(* IEC 61131-3 sources: NachHouse_CORE/V200/APP (part 3) *)

		r2	: NH_DAT_TIM2  := (txt:=                        	// zadanie datumu/casu
         [ (),(),(),(),(),(),(),(),
				(wh:=0),             										// ziadny text v urovni title
				(wh:=0)                         							// ziadny text pred datumom
			]);

      s  	: ARRAY[0..1] OF NH_SLD_DAT :=
         [  (t:=1,v1:=1, v2:=31, fmt := '%3.0f', txt:= 116, zom:=0,tun:=0),        										// 0 slider k start
				(t := 5,v1:=1,       v2 := 1439.0  , fmt := ''          , txt :=   0, xv := x2-53, tun := 1  )    // slider LUPY bodu, nevypisuje sa ani text, ani hodnota
         ];
   END_STRUCT;
  	NH_FRM_031  {HIDDEN} :    STRUCT     //31 FRM - ROM*set typ miestnosti
      hed : NH_FRM_HED := (Name:='_031',wht:=2,row:=1,sld:=0,desc:='Typ ROM');
      txt   : ARRAY[0..0] OF NH_OBJ_DAT :=
          [(wh:=6 , x:=xc,       y:= y1 + 60,  w:= 400, h:=28, Fgc:=4, fn:=2, nTch:=1, cf:=(n:=435))];           // typ miestosti

      mnu   : NH_OBJ_123 := // 2 riadky
            (wh:=123,cf:=(x:= 100,     y:= y1 + 130, typ:=2, rw2:=7, h:= 50, hTxt:= 28),
                 txt:=[436,437,438,439,440,441,511,512]);                                                    // 1 rolovaci vyber textov
      wrk   : ARRAY[3..10] OF NH_OBJ_DAT :=
          [(wh:= 0,   x:= xc , 		y:= y1 + 690, w:= 450, Fn := 2,  FgC :=5, BgC := 0, h := 24, cf:=(c:=0,n:=563), nTch:=1),	// 3 pouzit snimac osvelenia z
           (wh:=21,  x:= x2- 70 , 	y:= y1 + 550,  w:= 45, Fn :=563, FgC := 4, BgC := 50, h:=26),    	// 4 teplotu zo zony
           (wh:= 0,  x:= x2- 70 , 	y:= y1 + 600,  w:= 45, Fn :=564, FgC := 4, BgC := 50, h:=26),     // 5 osvetlenie z vonkajsej zony
           (wh:= 0,  x:= x2- 70 , 	y:= y1 + 650,  w:= 45, Fn :=565, FgC := 4, BgC := 50, h:=26),     // 6 osvetlenie z nadradenej zony
           (wh:=21,  x:= x2- 70 , 	y:= y1 + 700,  w:= 45, Fn :=566, FgC := 4, BgC := 50, h:=26),      // 7 CO2 zo zony
           (wh:= 0,  x:= x2- 70 , 	y:= y1 + 830,  w:= 45, Fn :=566, FgC := 4, BgC := 50, h:=26),
           (wh:= 0,  x:= x2- 70 , 	y:= y1 + 875,  w:= 45, Fn :=567, FgC := 4, BgC := 50, h:=26)
				// pred 3

			];

   END_STRUCT

//   NH_ZON_SET  {HIDDEN} : STRUCT      // ROM typ miestnosti
  	NH_FRM_032  {HIDDEN} :    STRUCT              //32 FRM - ZON*Set typ zony ....
      hed : NH_FRM_HED := (Name:='_032',wht:=2,row:=1,sld:=0,desc:='Typ ZON');

      txt   : ARRAY[0..0] OF NH_OBJ_DAT :=
          [ (wh:=6 , x:=xc,       y:= y1 + 60,  w:= 400, h:=28, Fgc:=4, fn:=2, nTch:=1, cf:=(n:=442))];           // typ miestosti
      mnu   : NH_OBJ_123 := // 2 riadky
            (wh:=123,cf:=(x:= 100,     y:= y1 + 130, typ:=2, rw2:=5, h:= 50, hTxt:= 28),
                 txt:=[443,444,445,446,447]);                                                    // 1 rolovaci vyber textov
      wrk   : ARRAY[3..10] OF NH_OBJ_DAT :=
          [(wh:= 0,  x:= xc , 		y:= y1 + 690, w:= 450, Fn := 2,  FgC :=5, BgC := 0, h := 24, cf:=(c:=0,n:=563), nTch:=1),	// 3 pouzit snimac osvelenia z
           (wh:= 0,  x:= x2- 70 , 	y:= y1 + 740,  w:= 45, Fn :=564, FgC := 4, BgC := 50, h:=22),                                    // 4
           (wh:= 0,  x:= x2- 70 , 	y:= y1 + 785,  w:= 45, Fn :=565, FgC := 4, BgC := 50, h:=22),
           (wh:= 0,  x:= x2- 70 , 	y:= y1 + 830,  w:= 45, Fn :=566, FgC := 4, BgC := 50, h:=22),
           (wh:= 0,  x:= x2- 70 , 	y:= y1 + 875,  w:= 45, Fn :=567, FgC := 4, BgC := 50, h:=22)
			];
   END_STRUCT

   NH_FRM_033  {HIDDEN} :  STRUCT 	// FRM - predvlby teploty
      hed : NH_FRM_HED := (Name:='_033',wht:=2,row:=1,sld:=5);
		PV_0_2			: ARRAY[0..2] OF NH_OBJ_DAT;
 		TX2				: NH_OBJ_DAT :=
		 		(wh:=6,  x:= x2/2   , 	y:= y1 +250, w:= 400,FgC := 4, BgC := 0, fn := 2, 	h:=33,cf:=(n:=592));   		// predvolby reguluju
		PV_4_10			: ARRAY[4..10] OF NH_OBJ_DAT;

      PV_SLD_XXX  	: ARRAY[0..4] OF NH_SLD_DAT :=  // definica a nazvy sliderov
         [  (t:=0,	xv := x2-53, v1 := 0.0, v2 :=100.0 , fmt := '%5.0f %%'       			   ,txt:= 83 ),     // 0 off       	txt:=cislo textu
            (t:=0,	xv := x2-53, v1 := 0.0, v2 :=100.0 , fmt := '%5.0f %%'      			   ,txt:= 154),     // 1 Minimum
            (t:=0,	xv := x2-53, v1 := 0.0, v2 :=100.0 , fmt := '%5.0f %%'      			   ,txt:= 156),     // 2 Normal
            (t:=0,	xv := x2-53, v1 := 0.0, v2 :=100.0 , fmt := '%5.0f %%'						,txt:= 165),     // 3 Maximum
            (t:=1, 	xv := x2-53, v2 :=255.0, 				 fmt := 's%Tm:ss m'						,txt:= 190) 	  // 4 opozdenie technologie
			];

   END_STRUCT;

	NH_FRM_035  {HIDDEN}  :  STRUCT 	//
      hed : NH_FRM_HED := (Name:='_035',desc:='FRM-TER/TEH/TEK Stp',wht:=2,row:=1,sld:=4);
      r  : ARRAY[1..1] OF NH_ROW_O := [( ob := [
            (wh:=221,x:= 50	,y:= y1 + 100, w:= 25 , 	h := 30,  	FgC :=10, BgC := 5,	Fn :=132,),     			// 0 hodnota zo snimaca
            (wh:=13, x:= 50   ,y:= y1 + 220, w:= x2-110, h := 251,	FgC := 4, BgC := 3, 	fn := 0),            	// 1 Korekcia - Konverzý faktor
            (wh:=221,x:= 50	,y:= y1 + 310, w:= 25 , 	h := 30,  	FgC := 3, BgC := 5, 	fn :=149,),          	// 2 hodnota po korekcii
           	(),
            (),
            (),
            (wh:=13, x:= 50   ,y:= y1 + 500, w:= x2-110 , h := 251,	FgC := 4, BgC := 2, 	fn := 1),              	// 6 povolena zmena
            (wh:=13, x:= 50   ,y:= y1 + 600, w:= x2-110 , h := 251,	FgC := 4, BgC := 2, 	fn := 2),              	// 7 opozdnie zmeny
            (wh:=13, x:= 50   ,y:= y1 + 700, w:= x2-110 , h := 251,	FgC := 4, BgC := 2, 	fn := 3),              	// 8
			   (wh:=20, x:=x2-60 ,y:= y1 + 820, w:= 48     , 				FgC := 0, BgC :=50, 	fn := 241),	  				// 9 neposielat do room
			   (wh:=20, x:=x2-60 ,y:= y1 + 880, w:= 48     , 				FgC := 4, BgC :=50, 	fn := 100)  				//10 zablokovat

       )];
      s  : ARRAY[0..3] OF NH_SLD_DAT := [
            ( t:=0, xv := x2-53, v1:=-20.0, 	v2 := 20.0 ,  fmt := '%+5.1f °C',   txt:= 119, ink:=0.1),      	// 0 Korekcia - Konverzý faktor
            ( t:=0, xv := x2-53, v1:=0.0, 	v2 := 10.0 ,  fmt := '%5.1f', 		txt:= 121, ink:=0.1),			// 1 povolena zmena
            ( t:=1, xv := x2-53, v1:=0.0, 	v2 := 254.0 , fmt := '%5.0f',   		txt:= 122),      					// 2 opozdenie zmeny
            ( t:=3, xv := x2-53, v1:=0.0, 	v2 := 3600.0, fmt := 's%Th:mm:ss h', 	txt:= 609)       					// 3 odoberat vzorky
			];
   END_STRUCT;

   NH_FRM_036 {HIDDEN}  :  STRUCT
      hed      : NH_FRM_HED := (Name:='_036',wht:=3);
      mnu      : NH_MNU := ( n:= 3,        // 7 MNU - TVE/VEN
                        o := [
                              (fn :=  6,wh:=   0,cm := 136),       		// < 1
                              (fn := 183,wh:= 25,cm :=   0),       		// 2
                              (fn := 344,wh:=345,cm := 205, frm:=33),  	// 3-predvolby
                              (fn := 220,wh:=221,cm := 205, frm:=30),   // 4 manual
                              (fn :=   0,wh:=191,cm :=   0, frm:= 0),   // 5-auto
                              (fn := 369,wh:=370,cm := 205, frm:=38), 	// 6-ochrana pred teplotou
	                           (fn := 348,wh:=348,cm :=  82),        		// 7-Rom, ktore vstupuu do ZON
                              (fn :=  23,wh:= 24,cm := 205, frm:=37)    // 8-setup TVE

                           ]);
   END_STRUCT;

   NH_FRM_037  {HIDDEN} : STRUCT      // TVE setup
      hed      : NH_FRM_HED := (Name:='_037',wht:=2,row:=1,sld:=2);
      mnu   : NH_OBJ_123 := // 2 riadky
            (wh:=123,cf:=(x:= 60,     y:= y1 + 80, typ:=2, rw2:=6, h:= 50, hTxt:= 28),
                 txt:=[466,467,468,469,470,471]);                                                    // 1 rolovaci vyber textov
      ROW   : ARRAY[2..10] OF NH_OBJ_DAT :=
            [(wh:=20, x:= x2-60  , y:= y1 + 400,   w:= 48     , FgC := 0, BgC :=50, fn := 171),            	// 2 NO/NC - inv
				 (wh:=0, x:= x2-60  , y:= y1 + 450,   w:= 48     , FgC := 0, BgC :=50, fn := 419),   				// 3 Analog
				 (wh:=20, x:= x2-60  , y:= y1 + 450,   w:= 48     , FgC := 0, BgC :=50, fn := 434),            	// 4 PWM
             (wh:=13, x:= 50     , y:= y1 + 600,   w:= x2-110 , FgC := 4, BgC := 3, fn := 0),              // 5 cas otvorenia
             (wh:=13, x:= 50     , y:= y1 + 680,   w:= x2-110 , FgC := 4, BgC := 3, fn := 1),              // 6 opozdenie technologie
				 (wh:=20, x:= x2-60  , y:= y1 + 750,   w:= 48     , FgC := 0, BgC :=50          , fn := 228 ), // 7 Log
             (wh:=20, x:= x2-60  , y:= y1 + 800,   w:= 48     , FgC := 4, BgC :=50			  	, fn := 100	), // 8 zablokovat
             (wh:=20, x:= x2-60  , y:= y1 + 860,   w:= 48     , FgC := 0, BgC :=50          , fn := 400 ) 	// 9 Externe DEV
		      ];
   	s  : ARRAY[0..1] OF NH_SLD_DAT := [
            ( t:=3, xv := x2-53, v2 :=  300.0 , fmt := 's%Tm:ss m',txt:= 167 ),      // 0 Cas otvorenia ventilu
            ( t:=1, xv := x2-53, v2 :=255.0 	 , fmt := 's%Tm:ss m',txt:= 190)   // 1 opozdenie technologie
         ];
   END_STRUCT

   NH_FRM_038  {HIDDEN}  :  STRUCT 	// FRM - predolby teploty
      hed      : NH_FRM_HED := (Name:='_038',wht:=2,row:=1,sld:=7);
      r  : ARRAY[1..1] OF NH_ROW_O := [( ob := [
				(wh:=21, x:= x2-70  , y:= y1 + 60,  w:= 45, Fn :=598, FgC := 4, BgC := 50, 	h:=28),			 	// 0 zapnut tepelnu ochanu

           	(wh:=6 , x:=xc,       y:= y1 + 160,  w:= 400, h:=28, Fgc:=4, fn:=2, nTch:=1, cf:=(n:=47)),   	// 1 Teplotna ochrana-kurenie
            (wh:=13, x:= 50     , y:= y1 + 300,   w:= x2-110 , FgC := 4, BgC := 3, fn := 0),              	// 2 min teplota
            (wh:=13, x:= 50     , y:= y1 + 380,   w:= x2-110 , FgC := 4, BgC := 18, fn := 1),              	// 3 max.teplotoa
            (wh:=13, x:= 50     , y:= y1 + 460,   w:= x2-110 , FgC := 4, BgC := 8, fn := 2),              	// 4 Optimalna teplota - zelena

	  			(wh:=6 , x:=xc,       y:= y1 + 570,  w:= 400, h:=28, Fgc:=4, fn:=2, nTch:=1, cf:=(n:=580)),  	// 5 Teplotna ochrana-chladenie
            (wh:=13, x:= 50     , y:= y1 + 700,   w:= x2-110 , FgC := 4, BgC := 3, fn := 3),              	// 6 min teplota
            (wh:=13, x:= 50     , y:= y1 + 780,   w:= x2-110 , FgC := 4, BgC :=18, fn := 4),              	// 7 max.teplotoa
            (wh:=13, x:= 50     , y:= y1 + 900,   w:= x2-110 , FgC := 4, BgC := 3, fn := 6)             		// 8 max cas zapnutia

       )];
      s  : ARRAY[0..6] OF NH_SLD_DAT := [
            ( t:=1, xv := x2-53, v2 := 130.0 , fmt := '%5.0f°',   txt:= 169),      // 0 min.teplota
            ( t:=1, xv := x2-53, v2 := 130.0 , fmt := '%5.0f°',   txt:= 170),      // 1 max.teplota
            ( t:=1, xv := x2-53, v2 := 130.0 , fmt := '%5.0f°',   txt:= 110),      // 2 udrziavacia teplota
            ( t:=1, xv := x2-53, v2 := 30.0 , fmt := '%5.0f°',   txt:= 169),      // 3 Min
            ( t:=1, xv := x2-53, v2 := 30.0 , fmt := '%5.0f°',   txt:= 170),      // 4 Max
            ( t:=1, xv := x2-53, v2 := 130.0 , fmt := '%5.0f°',   txt:= 110),      // 5

            ( t:=3, xv := x2-53, v2 := 2880.0 , fmt := 'm%Th:mm h',txt:=  62)      // 6 MAx.cas zapnutia
         ];
   END_STRUCT;

   NH_FRM_039 {HIDDEN}:  STRUCT 	//39 FRM - LED WSB/TGL
      hed      : NH_FRM_HED := (Name:='_039',wht:=2,row:=2,sld:=8,desc:='FRM-LED:WSB/TGL');
      r  : ARRAY[1..2] OF NH_ROW_O := [( ob := [
            (wh:=13, x:= 50     , y:= y1 + 100,   w:= x2-110  ,FgC := 4, BgC := 5,h:=251   , fn := 0             ), // Den-intensita
            (wh:=13, x:= 50     , y:= y1 + 180,   w:= x2-110  ,FgC := 4, BgC := 3,h:=251   , fn := 1             ), // 253 znamena, ze zmenu slidera bude ukladat do nejakej BOOL premennej
            (wh:=13, x:= 50     , y:= y1 + 260,   w:= x2-110  ,FgC := 4, BgC := 9,h:=251   , fn := 2             ),
            (wh:=13, x:= 50     , y:= y1 + 340,   w:= x2-110  ,FgC := 4, BgC := 8,h:=251   , fn := 3             ),
            (wh:=13, x:= 50     , y:= y1 + 470,   w:= x2-110  ,FgC := 4, BgC := 5,h:=251   , fn := 4             ), // Den-cas uspatia
            (wh:=13, x:= 50     , y:= y1 + 550,   w:= x2-110  ,FgC := 4, BgC := 3,h:=251   , fn := 5             ),
            (wh:=13, x:= 50     , y:= y1 + 630,   w:= x2-110  ,FgC := 4, BgC := 9,h:=251   , fn := 6             ),
            (wh:=13, x:= 50     , y:= y1 + 710,   w:= x2-110  ,FgC := 4, BgC := 8,h:=251   , fn := 7             ),
//            (wh:= 0, x:= x2/2   , y:= y1 + 380,   w:= 400    , FgC := 2, fn := 2, h:=25, cf:=(n:=139),nTch:=1    ),  // 'Uspat po case'
            (wh:=20, x:= x2-60  , y:= y1 + 770,   w:= 48, Fn :=480,  FgC :=10, BgC := 50, h := 0, cf :=(c:=3), cm:=140  ),  // 8 LED nad funcnym tlacitkom
            (wh:=20, x:= x2-60  , y:= y1 + 830,   w:= 48     , FgC := 0, BgC :=50          , fn := 55            ),  // 9  pohyb resetuje cas
            (wh:=20, x:= x2-60  , y:= y1 + 880,   w:= 48     , FgC := 0, BgC :=50          , fn := 111           )   //10  zobudit pohybom
              ]), ( ob := [
            (wh:= 6, x:= x2/2   , y:= y1 +  40,   w:= 400    , FgC := 2, fn := 2, h:=25, cf:=(n:=137),nTch:=1    ),   // 'Svietivost'
            (wh:= 6, x:= x2/2   , y:= y1 + 410,   w:= 400    , FgC := 2, fn := 2, h:=25, cf:=(n:=139),nTch:=1    )  // 'Uspat po case'
              )];
      s  : ARRAY[0..7] OF NH_SLD_DAT :=
           [
            (t := 1,                fmt := '%3.0f %%'            , txt:= 28),        // 0 Den - intenzita
            (t := 1,                fmt := '%3.0f %%'            , txt:= 29),        // 1 Vecr
            (t := 1,                fmt := '%3.0f %%'            , txt:= 30),        // 2 Noc
            (t := 1,                fmt := '%3.0f %%'            , txt:= 31),        // 3 Rano
            (t := 1, v2 := 238.0  , fmt := '3%Tm:ss m'           , txt:= 28),        // 4 Den - zas vypnutia
            (t := 1, v2 := 238.0  , fmt := '3%Tm:ss m'           , txt:= 29),        // 5 Vecr
            (t := 1, v2 := 238.0  , fmt := '3%Tm:ss m'           , txt:= 30),        // 6 Noc
            (t := 1, v2 := 238.0  , fmt := '3%Tm:ss m'           , txt:= 31)         // 7 Rano

              ];

   END_STRUCT;

   NH_FRM_057 {HIDDEN}:  STRUCT 	//39 FRM - LED WSB/TGL
      hed      : NH_FRM_HED := (Name:='_057',wht:=2,row:=2,sld:=8,desc:='FRM-TGL-casy uspatia');
      r  : ARRAY[1..2] OF NH_ROW_O := [( ob := [
            (wh:=13, x:= 50     , y:= y1 + 100,   w:= x2-110  ,FgC := 4, BgC := 5,h:=251   , fn := 0             ), // Den-intensita
            (wh:=13, x:= 50     , y:= y1 + 180,   w:= x2-110  ,FgC := 4, BgC := 3,h:=251   , fn := 1             ), // 253 znamena, ze zmenu slidera bude ukladat do nejakej BOOL premennej
            (wh:=13, x:= 50     , y:= y1 + 260,   w:= x2-110  ,FgC := 4, BgC := 9,h:=251   , fn := 2             ),
            (wh:=13, x:= 50     , y:= y1 + 340,   w:= x2-110  ,FgC := 4, BgC := 8,h:=251   , fn := 3             ),
            (wh:=13, x:= 50     , y:= y1 + 470,   w:= x2-110  ,FgC := 4, BgC := 5,h:=251   , fn := 4             ), // Den-cas uspatia
            (wh:=13, x:= 50     , y:= y1 + 550,   w:= x2-110  ,FgC := 4, BgC := 3,h:=251   , fn := 5             ),
            (wh:=13, x:= 50     , y:= y1 + 630,   w:= x2-110  ,FgC := 4, BgC := 9,h:=251   , fn := 6             ),
            (wh:=13, x:= 50     , y:= y1 + 710,   w:= x2-110  ,FgC := 4, BgC := 8,h:=251   , fn := 7             ),
//            (wh:= 0, x:= x2/2   , y:= y1 + 380,   w:= 400    , FgC := 2, fn := 2, h:=25, cf:=(n:=139),nTch:=1    ),  // 'Uspat po case'
            (wh:=20, x:= x2-60  , y:= y1 + 770,   w:= 48, Fn :=480,  FgC :=10, BgC := 50, h := 0, cf :=(c:=3), cm:=140  ),  // 8 LED nad funcnym tlacitkom
            (wh:=20, x:= x2-60  , y:= y1 + 830,   w:= 48     , FgC := 0, BgC :=50          , fn := 55            ),  // 9  pohyb resetuje cas
            (wh:=20, x:= x2-60  , y:= y1 + 880,   w:= 48     , FgC := 0, BgC :=50          , fn := 111           )   //10  zobudit pohybom
              ]), ( ob := [
            (wh:= 6, x:= x2/2   , y:= y1 +  40,   w:= 400    , FgC := 2, fn := 2, h:=25, cf:=(n:=137),nTch:=1    ),   // 'Svietivost'
            (wh:= 6, x:= x2/2   , y:= y1 + 410,   w:= 400    , FgC := 2, fn := 2, h:=25, cf:=(n:=139),nTch:=1    )  // 'Uspat po case'
              )];
      s  : ARRAY[0..7] OF NH_SLD_DAT :=
           [
            (t := 1,                fmt := '%3.0f %%'            , txt:= 28),        // 0 Den - intenzita
            (t := 1,                fmt := '%3.0f %%'            , txt:= 29),        // 1 Vecr
            (t := 1,                fmt := '%3.0f %%'            , txt:= 30),        // 2 Noc
            (t := 1,                fmt := '%3.0f %%'            , txt:= 31),        // 3 Rano
            (t := 1, v2 := 238.0  , fmt := '3%Tm:ss m'           , txt:= 28),        // 4 Den - zas vypnutia
            (t := 1, v2 := 238.0  , fmt := '3%Tm:ss m'           , txt:= 29),        // 5 Vecr
            (t := 1, v2 := 238.0  , fmt := '3%Tm:ss m'           , txt:= 30),        // 6 Noc
            (t := 1, v2 := 238.0  , fmt := '3%Tm:ss m'           , txt:= 31)         // 7 Rano

              ];

   END_STRUCT;

   NH_FRM_040  {HIDDEN} :  STRUCT 	// FRM - BLIKAC-jedna seria
      hed      : NH_FRM_HED := (Name:='_040',wht:=2,row:=1,sld:=7);
      r  : ARRAY[1..1] OF NH_ROW_O := [( ob := [
            (wh:=13, x:= 50     , y:= y1 + 100,   w:= x2-110  ,FgC := 4, BgC := 5          , fn := 0             ), // 0 Pocet bliknuti
            (wh:=13, x:= 50     , y:= y1 + 200,   w:= x2-110  ,FgC := 4, BgC := 3          , fn := 4             ), // 1 Cas ON
            (wh:=13, x:= 50     , y:= y1 + 300,   w:= x2-110  ,FgC := 4, BgC := 3          , fn := 5             ), // 2 Cas OFF
            (wh:=20, x:= x2-60  , y:= y1 + 380,   w:= 48     , FgC := 0, BgC :=50          , fn := 399           ), // 3 rovnaka uroven
            (wh:=13, x:= 50     , y:= y1 + 480,   w:= x2-110  ,FgC := 4, BgC := 5          , fn := 1             ), // 4 Lvl ON
            (wh:=13, x:= 50     , y:= y1 + 560,   w:= x2-110  ,FgC := 4, BgC := 5          , fn := 2             ), // 5 Lvl OFF
            (wh:=13, x:= 50     , y:= y1 + 640,   w:= x2-110  ,FgC := 4, BgC := 5          , fn := 3             ), // 6 rampa
            (wh:=13, x:= 50     , y:= y1 + 780,   w:= x2-110  ,FgC := 4, BgC := 2          , fn := 6             ), // 7 Odlozenie startu
            (wh:=20, x:= x2-60  , y:= y1 + 835,   w:= 48     , FgC := 0, BgC :=50          , fn := 59            ), // 8  Po startom vypnut
            (wh:=20, x:= x2-60  , y:= y1 + 885,   w:= 48     , FgC := 0, BgC :=50          , fn := 60            )  // 9  Na konci vypnut

              )];
      s  : ARRAY[0..6] OF NH_SLD_DAT :=
           [
            (t := 1, v1:=1.0, v2:=255.0,  fmt := '%3.0f'          , txt:= 86),                  // 0 pocet bliknuti
            (t := 1,                      fmt := '%3.0f %%'       , txt:=252),                  // 1 lvl-ON
            (t := 1,                      fmt := '%3.0f %%'       , txt:=253),                  // 2 lvl-OFF
            (t := 1,          V2:=15.0,   fmt := '%2.0f'          , txt:=364),                  // 3 rampa
            (t := 3,          v2:= 1200.0,fmt := '5%Tm:ss.zz m'   , txt:= 87,ink:=1.0),       // 4 t-On
            (t := 3,          v2:= 1200.0,fmt := '5%Tm:ss.zz m'   , txt:= 88,ink:=1.0),       // 5 t-Off
            (t := 3,          v2:= 3000.0,fmt := '1%Tm:ss.z m'    , txt:=73, ink:=1.0)          // 6 Odlozenie startu
              ];
   END_STRUCT;

   NH_FRM_041 {HIDDEN}  :  STRUCT
      hed      : NH_FRM_HED := (Name:='_041',wht:=3);
      mnu      : NH_MNU := ( n:= 3,                                // nastavenie parMWTROV
                        o := [
                              (fn :=   6,wh:=  6,cm :=  31),
                              (),
                              (fn :=  83,wh:= 84,cm := 205,x:=xc-90  ,frm:=40),       // par.bliknutie jednej serie
                              (fn := 196,wh:=197,cm := 205,x:=xc	  ,frm:=42),        // pocet serii
										(fn := 348,wh:=348,cm :=  82,x:=xc+90				)			// ROM->DEV
                           ]);
   END_STRUCT;

   NH_FRM_042 {HIDDEN}  :  STRUCT 	// FRM - BLIKAC-pocet serii
      hed      : NH_FRM_HED := (Name:='_042',wht:=2,row:=1,sld:=5);
      r  : ARRAY[1..1] OF NH_ROW_O := [( ob := [
            (wh:=13, x:= 50     , y:= y1 + 150,   w:= x2-110  ,FgC := 4, BgC := 5          , fn := 0             ), // 0 Pocet serii
            (wh:=13, x:= 50     , y:= y1 + 250,   w:= x2-110  ,FgC := 4, BgC := 3          , fn := 1             ), // 1 LVL do dalse serie
            (wh:=13, x:= 50     , y:= y1 + 350,   w:= x2-110  ,FgC := 4, BgC := 3          , fn := 2             ), // 2 LVL do dalse serie
            (wh:=13, x:= 50     , y:= y1 + 500,   w:= x2-110  ,FgC := 4, BgC := 2          , fn := 3             )  // 3 max cas
              )];
      s  : ARRAY[0..4] OF NH_SLD_DAT :=
           [
            (t := 1, v1:=1.0, v2:=255.0,  fmt := '%3.0f'          , txt:= 89),               // 0 pocet serii
            (t := 1,                      fmt := '%3.0f %%'       , txt:=397),               // 1 lvl- Next serie
            (t := 3,          v2:=36000.0,fmt := 's%Th:mm:ss h'   , txt:=398,ink:=1.0),     // 2 t-cakanie do dalsej serie
            (t := 3, v1:=0.0, v2:= 1440.0,fmt := 'm%Th:mm h'      , txt:=62,ink:=1.0)        // 3 max.cas zapnutia

              ];
   END_STRUCT;

  	NH_FRM_043  {HIDDEN} :    STRUCT               // BRW:  SVD,SVA,RGB,ZAS,SIR,DOR,WIN,
      hed      : NH_FRM_HED := (Name:='_043',wht:=1,row:=3,sld:=3);
      D1_1_4      : NH_brw_D1_ALL;                          // 0..4 : podklad/dev/stat/fav/
      D1_5_SLD    : NH_brw_D1_SLD;   				// 5=slider
      D1_6_PIR    : NH_brw_D1_PIR;	//ARRAY[6..6] OF NH_OBJ_DAT ;
//      D1_7        : NH_OBJ_4O := (wh:= 0, obj:=1, ok:=[1,0,0,1], crc:=[1,1,1,1], FgT:= [1,1,4,1], BgC:=[10,7,7,10],  txt:=[1,0,1,1], obr:=[0,0,0,1] );                // 8 = time/blkPIR na dstavom
//      D1_8        : NH_OBJ_4O := (wh:=107, obj:=2, ok:=[1,1,0,0], crc:=[1,0,1,1], FgT:= [1,1,4,1], BgC:=[10,0,7,10], txt:=[1,0,1,1], wxy :=[34,34,34,34] ), cm:=[44];  // 8 = time/blkPIR na dstavom
      D1_7        : NH_OBJ_4O1 := (wh:=0);              														// 7 = DayMode/Sviecka
      D1_8        : NH_OBJ_4O2;	// := (wh:=107, obj:=2, cmd :=[44,45], FgT:= [1,1,4,1], BgC:=[10,0,7,10]);       // 8 = Time-OFF/BlokPir
      D1_9_10NAZ  : NH_brw_D1_NAZ;                                // 9..10 Nazov rom + DEV

      D2  : NH_ROW_O_D1;       // dash 2
      D3  : NH_ROW_O_D1;       // dash 3

      SL : NH_brw_SLD;
   END_STRUCT;

   NH_FRM_044  {HIDDEN} :  STRUCT 	// FRM - setup SVD,SVA,ZAS,SIR
      hed      : NH_FRM_HED := (Name:='_044',wht:=2,row:=1,sld:=6);
      r  : ARRAY[1..1] OF NH_ROW_O := [( ob := [
            (wh:=20, x:= x2-60  , y:= y1 +  60,   w:= 48     , FgC := 4, BgC :=50          , fn := 100          ), // 0 zablokovat
            (wh:=20, x:= x2-60  , y:= y1 + 110,   w:= 48     , FgC := 0, BgC :=50          , fn := 106          ), // 1 Inverzna funkcia
            (wh:=20, x:= x2-60  , y:= y1 + 860,   w:= 48     , FgC := 0, BgC :=50          , fn := 400          ), // 2 Externe DEV
            (wh:=20, x:= x2-60  , y:= y1 + 160,   w:= 48     , FgC := 0, BgC :=50          , fn := 146          ), // 3 Obnovit LVL po restarte
            (wh:=13, x:= 50     , y:= y1 + 260,   w:= x2-110  ,FgC := 4, BgC := 5          , fn := 0            ), // 4 Prikon
            (wh:=13, x:= 50     , y:= y1 + 350,   w:= x2-110  ,FgC := 4, BgC := 3          , fn := 1            ), // 5 Stmievatelne minimum
            (wh:=13, x:= 50     , y:= y1 + 440,   w:= x2-110  ,FgC := 4, BgC := 3          , fn := 2            ), // 6 Efektivne maximum
            (wh:=20, x:= x2-60  , y:= y1 + 520,   w:= 48     , FgC := 0, BgC :=50          , fn := 153          ), // 7 Vlastne stmievani
            (wh:= 0, x:= 50     , y:= y1 + 620,   w:= x2-110  ,FgC := 4, BgC := 3          , fn := 3            ), // 8 krok stmievania Fade Rate
            (wh:= 0, x:= 50     , y:= y1 + 700,   w:= x2-110  ,FgC := 4, BgC := 3          , fn := 4            ), // 9 Fade Time
            (wh:=13, x:= 50     , y:= y1 + 800,   w:= x2-110  ,FgC := 4, BgC := 2          , fn := 5            ) //10 opozdene zazatie  po vypnuti
              )];
      s  : ARRAY[0..5] OF NH_SLD_DAT :=
           [
            (t := 0,      		v2:= 3000.0 , fmt := '%4.0f W'            , txt:=  69),        // 0 Prikon
            (t := 1                       , fmt := '%3.0f %%'       		, txt:=  70),      	// 1 stmievatelne minimum
            (t := 1                       , fmt := '%3.0f %%'       		, txt:=  71),       	// 2 efektivma maximum
            (t := 1, v1:=1.0, v2:=10      , fmt := '%3.0f'        		, txt:= 365),       	// 3 krok stmievania Fade Rate
            (t := 1, v1:=1.0, v2:=10      , fmt := '%3.0f'         		, txt:= 364),       	// 4 Fade Time
            (t := 1,          v2:=50.0 	, fmt := '1%Ts.z s'           , txt:= 145)        	// 5 opozdene zazati  po vypnuti
              ];
   END_STRUCT;
   NH_FRM_045 {HIDDEN}  :  STRUCT
      hed      : NH_FRM_HED := (Name:='_045',wht:=3);
      mnu      : NH_MNU := ( n:=3,                                  // MNU-SVD,SVA,SCN
                        o := [
                              (fn :=   6,wh:=  6,cm :=  31),
                              (),
                              (fn :=  83,wh:= 84,cm := 205,x:=xc-90 	,frm:=9	),        // parametre
                              (fn :=  23,wh:= 24,cm := 205,x:=xc		,frm:=44	),        // setup
										(fn := 348,wh:=348,cm :=  82,x:=xc+90				),        // ROM ->
										(fn :=   0,wh:= 73,cm := 205,x:=xc+180,frm:=91  )         // typ ZAS
                           ]);
   END_STRUCT;
   NH_FRM_046 {HIDDEN}  :  STRUCT
      hed      : NH_FRM_HED := (Name:='_046',wht:=3);
      mnu      : NH_MNU := ( n:=3,                                  // MNU-SVD,SVA,
                        o := [
                              (fn :=   6,wh:=  6,cm :=  31),
                              (),
                              (fn :=  83,wh:= 84,cm := 205,x:=xc-135 	,frm:= 9),        // parametre
                              (fn := 124,wh:=125,cm := 205,x:=xc-45  	,frm:=47),        // RGB
										(fn := 348,wh:=348,cm :=  82,x:=xc+45			  ),			// ROM->DEV
                              (fn :=  23,wh:= 24,cm := 205,x:=xc+135 	,frm:=44)        // setup
                           ]);
   END_STRUCT;

   NH_FRM_047 {HIDDEN}  :  STRUCT 	// FRM - RGB
      hed      : NH_FRM_HED := (Name:='_047',wht:=2,row:=1,sld:=5);
      r  : ARRAY[1..1] OF NH_ROW_O := [( ob := [
				(wh:=0),
            (wh:=112, x:= xc-5  , y:= y1 + 280,   w:= 500, fn := 126, prs:=true),      										// 1 RGB obrazok 6/1
            (wh:=113, x:= 100   , y:= y1 + 590,   w:= 800, fn := 42, h:= 42, prs :=true  	            ), 	// 2 predvolby
            (wh:=13, x:= 50     , y:= y1 + 660,   w:= x2-200  ,FgC := 7, BgC := 7, h := 8 , fn := 0            ), 	// 3 R
            (wh:=13, x:= 50     , y:= y1 + 720,   w:= x2-200  ,FgC := 8, BgC := 8, h := 8 , fn := 1            ), 	// 4 G
            (wh:=13, x:= 50     , y:= y1 + 780,   w:= x2-200  ,FgC := 9, BgC := 9, h := 8 , fn := 2            ), 	// 5 B
            (wh:=13, x:= 50     , y:= y1 + 840,   w:= x2-200  ,FgC := 4, BgC := 4, h := 8 , fn := 3            ), 	// 6 CW
            (wh:=13, x:= 50     , y:= y1 + 900,   w:= x2-200  ,FgC :=30, BgC :=30, h := 8 , fn := 4            ),	 	// 7 WW - amber
            (wh:= 0, x:= 50     , y:= y1 + 700,   w:= x2-110  ,FgC := 4, BgC := 3         , fn := 4            ), 	// 8
            (wh:= 0, x:= 50     , y:= y1 + 800,   w:= x2-110  ,FgC := 4, BgC := 2         , fn := 5            ) 	// 9
              )];
      s  : ARRAY[0..5] OF NH_SLD_DAT :=
           [

            (t := 1, v2 := 255.0  , fmt := '>%3.0f', zom := 0 ),        // 0 R
            (t := 1, v2 := 255.0  , fmt := '>%3.0f', zom := 0 ),        // 1 G
            (t := 1, v2 := 255.0  , fmt := '>%3.0f', zom := 0 ),        // 2 B
            (t := 1, v2 := 255.0  , fmt := '>%3.0f', zom := 0 ),        // 3 WW
            (t := 1, v2 := 255.0  , fmt := '>%3.0f', zom := 0 )         // 4 CW
              ];
   END_STRUCT;

	NH_FRM_048  {HIDDEN} :    STRUCT               // 5 BRW-dali-MASTER
      hed      : NH_FRM_HED := (Name:='_048',wht:=1,row:=3,sld:=3);
      D1_1_4     : NH_brw_D1_ALL;
		D1_1_6	  : NH_brw_D1_GATE;
      D1_6_SLD   : NH_brw_D1_SLD	:= ( ob := ( x := 170, w:=300, BgC:=7 ) );                          // 5=slider
      D1_7       : NH_OBJ_4O1 	:= (  wh:=0 );                          // 5=slider;
      D1_8       : NH_OBJ_4O2    := (  wh:=0 );
      D1_NAZ     : NH_brw_D1_NAZ;                          // 9..10 Nazov rom + DEV

      r  : ARRAY[1..2] OF NH_row_O_D1;

		SL : NH_brw_SLD;
   END_STRUCT;

   NH_FRM_049 {HIDDEN}  :  STRUCT
      hed      : NH_FRM_HED := (Name:='_049',wht:=3);
      mnu      : NH_MNU := ( n:=8,                                  // MNU-SVD,SVA,
                        o := [
                              (fn :=   6,wh:=  6,cm :=  31),
                              (),
                              (),
                              (),
                              (),
                              (),
                              (),
                              (fn :=  23,wh:= 24,cm := 205,x:=xc ,frm:=50)        // setup - default pre ALA
                           ]);
   END_STRUCT;

   NH_FRM_050  {HIDDEN} :  STRUCT 	// FRM - setup ALA
      hed      : NH_FRM_HED := (Name:='_050',wht:=2,row:=1,sld:=1);
      r  : ARRAY[1..1] OF NH_ROW_O := [( ob := [
            (wh:=20, x:= x2-60  , y:= y1 + 210,   w:= 48     , FgC := 0, BgC :=50          , fn := 450          ), // 1 Qr = prvy vstup podla LVL alarmu
            (wh:=20, x:= x2-60  , y:= y1 + 280,   w:= 48     , FgC := 0, BgC :=50          , fn := 451          ), // 2 pohyb
            (wh:=0,  x:= x2-60  , y:= y1 + 480,   w:= 48     , FgC := 0, BgC :=50          , fn := 453          ), // 4 Ostražitost ukoncena
            (wh:=0,  x:= x2-60  , y:= y1 + 560,   w:= 48     , FgC := 0, BgC :=50          , fn := 454          ), // 5 Stráženie obnovené
            (wh:=0, 	x:= x2-60  , y:= y1 + 510,   w:= 48     , FgC := 0, BgC :=50          , fn := 0            ), // 6
				(wh:=6 , x:= xc,      y:= y1 +  90,   w:= 500, h:= 28,  Fn := 2, FgC := 4,   cf:=(n:=449)),                      // 0 nazov: Tyzdenny program
            (wh:=13, x:= 50     , y:= y1 + 390,   w:= x2-110  ,FgC := 4, BgC := 5          , fn := 0            )  // 8 Filter pohybu
              )];
      s  : ARRAY[0..0] OF NH_SLD_DAT :=
           [
            (t := 3,      		v2:= 300.0 , fmt := 's%Tm:ss m'            , txt:=  452)        //
              ];

   END_STRUCT;

	NH_FRM_051 {HIDDEN}:  STRUCT 	// FRM parametre GATE
      hed      : NH_FRM_HED := (Name:='_051',wht:=2,row:=1,sld:=4);
      r  : ARRAY[0..0] OF NH_ROW_O := [( ob := [
            (wh:= 0, x:= 50     , y:= y1 + 100,   w:= x2-110  ,FgC := 4, BgC := 5          , fn := 0             ), // 0 otvorit na
            (wh:= 0, x:= 50     , y:= y1 + 200,   w:= x2-110  ,FgC := 4, BgC := 5          , fn := 1             ), // 1 vykonat s opozdenim
            (wh:= 0, x:= 50     , y:= y1 + 350,   w:= x2-110  ,FgC := 4, BgC := 3          , fn := 2             ), // 2 zatvorit po case
            (wh:= 0, x:= 50     , y:= y1 + 450,   w:= x2-110  ,FgC := 4, BgC := 3          , fn := 3             ), // 3 zatvorit po case pri lck
            (wh:= 0, x:= x2-60  , y:= y1 + 520,   w:= 48     , FgC := 0, BgC :=50          , fn := 55            ), // 4 pritomnost resetuje cas zatvorenia
            (wh:= 0, x:= x2-60  , y:= y1 + 800,   w:= 48     , FgC := 4, BgC :=50			  , fn := 100           ), // zablokovat
				(),
				(),
				(),
				(),
            (wh:= 0, x:=xc      , y:= 1015,       w:= 400, h:=20, Fgc:=2, fn:=2, nTch:=1, cf:=(c:=254)           )  // 10 info
				                                 )];
      s  : ARRAY[0..3] OF NH_SLD_DAT :=
           [
            (t := 1, v2 := 100.0, fmt := '%3.0f %%'            , txt:= 456),
            (t := 3, v2 := 60.0 , fmt := '%3.0f m'   	, txt:= 115),
            (t := 1, v2 := 60.0 , fmt := '%3.0f m'         		, txt:= 457),
            (t := 1, v2 := 60.0 , fmt := '%3.0f m'         		, txt:= 458)
              ];
   END_STRUCT;

	NH_FRM_052 {HIDDEN}:  STRUCT 	// FRM setup GATE
      hed      : NH_FRM_HED := (Name:='_052',wht:=2,row:=1,sld:=3);
      r  : ARRAY[0..0] OF NH_ROW_O := [( ob := [
            (wh:= 0, x:= 50     , y:= y1 + 100,   w:= x2-110  ,FgC := 4, BgC := 5          , fn := 0             ), // 0 cas impulzu
            (wh:= 0, x:= 50     , y:= y1 + 200,   w:= x2-110  ,FgC := 4, BgC := 3          , fn := 1             ), // 1 reverzny cas
            (wh:= 0, x:= 50     , y:= y1 + 300,   w:= x2-110  ,FgC := 4, BgC := 3          , fn := 2             ), // 2 cas otvorenia
            (wh:= 0, x:= 50     , y:= y1 + 400,   w:= x2-110  ,FgC := 4, BgC := 3          , fn := 3             ), // 3 cas zatvorenia
            (wh:= 0, x:= x2-60  , y:= y1 + 500,   w:= 48     , FgC := 0, BgC :=50          , fn := 117           ), // 4 pouzit HW koncovy snimac
            (wh:=20, x:= x2-60  , y:= y1 + 550,   w:= 48     , FgC := 0, BgC :=50          , fn := 124  	      ), // 5 Koncovy snimac su dvere
            (wh:= 0, x:= x2-60  , y:= y1 + 600,   w:= 48     , FgC := 0, BgC :=50          , fn := 465           ), // 6 samostatne rele Open/Close
            (wh:=20, x:= x2-60  , y:= y1 + 650,   w:= 48     , FgC := 0, BgC :=50          , fn := 461           ), // 7 rele open is real
            (wh:= 0, x:= x2-60  , y:= y1 + 700,   w:= 48     , FgC := 0, BgC :=50          , fn := 462           ), // 8 rele close is real
            (wh:=20, x:= x2-60  , y:= y1 + 800,   w:= 48     , FgC := 0, BgC :=50          , fn := 228           ), // 9 Log
            (wh:=20, x:= x2-60  , y:= y1 + 850,   w:= 48     , FgC := 4, BgC :=50			  , fn := 100           )  // 10 zablokovat

              )];
      s  : ARRAY[0..3] OF NH_SLD_DAT :=
           [
            (t := 1, v2 := 100.0    , fmt := '1%Ts:z s'          	, txt:= 116),
				(t := 1, v1:= 1, v2 := 100.0    , fmt := '1%Ts:z s'          	, txt:= 98),
            (t := 3, v2 := 1800.0 , fmt := '1%Tm:ss m'         	, txt:= 459),
            (t := 3, v2 := 1800.0 , fmt := '1%Tm:ss m'         	, txt:= 460)
              ];

   END_STRUCT;
   NH_FRM_053 {HIDDEN}  :  STRUCT
      hed      : NH_FRM_HED := (Name:='_053',desc:='MNU: ROM->DEV',wht:=3);
      mnu      : NH_MNU := ( n:=3,                                  				// MNU-GATE
                        o := [
                              (fn :=   6,wh:=  6,cm :=  31),
                              (),
                              (fn :=  83,wh:= 84,cm := 205,x:=xc-90 ,frm:=51),        // parametre
										(fn := 348,wh:=348,cm :=  82,x:=xc   			),			// ROM->DEV
                              (fn :=  23,wh:= 24,cm := 205,x:=xc+90 ,frm:=52)        // setup

                           ]);
   END_STRUCT;
   NH_FRM_054 {HIDDEN}  :  STRUCT
      hed      : NH_FRM_HED := (Name:='_054',wht:=3);
      mnu      : NH_MNU := ( n:=8,
									o := [		(fn :=   6,wh:=  0,cm :=  31),       // <
                                       (fn :=   0,wh:=  6,cm :=   0, w:=72),  // obrazok vyssej casti
                                       (fn :=  35,wh:= 38,cm :=  33),          // 3 check
                                       (),          										// 4 cat
                                       (),          										// 5 all.rom / 1rom
                                       (),          										// 6 priradit rom
                                       (),          										// 7-list
                                       (fn := 348,wh:=348,cm :=  82)]
											);
   END_STRUCT;

	NH_FRM_055 {HIDDEN}:  STRUCT 	// FRM cfg DOR,WIN,CO2...
      hed      : NH_FRM_HED := (Name:='_055',wht:=2,row:=1,sld:=3);
      r  : ARRAY[0..0] OF NH_ROW_O := [( ob := [
            (wh:=20, x:= x2-60  , y:= y1 + 100,   w:= 48     , FgC := 0, BgC :=50          , fn := 101           ), // 0 signal je pri rozopnuti
            (wh:=13, x:= 50     , y:= y1 + 230,   w:= x2-110  ,FgC := 4, BgC := 3          , fn := 0             ), // 1 znizenie citlivosti unLOCK
            (wh:=20, x:= x2-60  , y:= y1 + 300,   w:= 48     , FgC := 0, BgC :=50          , fn := 227           ), // 2 je sucastou alarm
            (wh:=13, x:= 50     , y:= y1 + 400,   w:= x2-110  ,FgC := 4, BgC := 3          , fn := 1             ), // 3 znizenie citlivosti LOCK
            (wh:=13, x:= 50     , y:= y1 + 500,   w:= x2-110  ,FgC := 4, BgC := 3          , fn := 2             ), // 4 OFF-autoreset
            (wh:=20, x:= x2-60  , y:= y1 + 600,   w:= 48     , FgC := 0, BgC :=50          , fn := 102           ), // 5 jeden tamper
            (wh:=20, x:= x2-60  , y:= y1 + 650,   w:= 48     , FgC := 0, BgC :=50          , fn := 103           ), // 6 dvojite vyvazenie
            (wh:=20, x:= x2-60  , y:= y1 + 750,   w:= 48     , FgC := 0, BgC :=50          , fn := 228           ), // 7 Log
            (wh:=20, x:= x2-60  , y:= y1 + 800,   w:= 48     , FgC := 4, BgC :=50			  , fn := 100			   ), // 8 zablokovat
            (wh:=20, x:= x2-60  , y:= y1 + 860,   w:= 48     , FgC := 0, BgC :=50          , fn := 400           ) 	// 9 Externe DEV
              )];
      s  : ARRAY[0..2] OF NH_SLD_DAT :=
           [
            (t := 1, v2 := 100.0  , fmt := '%3.0f'       		, txt:= 104),
            (t := 1, v2 := 100.0  , fmt := '%3.0f'       		, txt:= 463),
            (t := 3, v2 := 1800.0 , fmt := 's%Tm:ss m'         , txt:= 464)
              ];

   END_STRUCT;
   NH_FRM_056 {HIDDEN}  :  STRUCT
      hed      : NH_FRM_HED := (Name:='_056',wht:=3);
      mnu      : NH_MNU := ( n:=3,                                  // MNU-SVD,SVA,SCN
                        o := [
                              (fn :=   6,wh:=  6,cm :=  31),
                              (w:=72),
                              (fn :=  23,wh:= 24,cm := 205,x:=xc-45	,frm:=55	), 	// 3 setup
										(fn := 348,wh:=348,cm :=  82,x:=xc+45				)		// 4 ROM->DEV
                           ]);
   END_STRUCT;

	NH_FRM_058  {HIDDEN}  :  STRUCT 	// FRM - tune LUX,CO2,CO...
      hed      : NH_FRM_HED := (Name:='_058',wht:=2,row:=1,sld:=6);
      r  : ARRAY[1..1] OF NH_ROW_O := [( ob := [
            (wh:=221,x:= 50	,y:= y1 +  60, w:= 25 , 	h := 33,  	FgC := 4, BgC := 5,	Fn :=132,),     			// 0 hodnota zo snimaca
            (wh:=13, x:= 50   ,y:= y1 + 170, w:= x2-110, h :=251,		FgC := 4, BgC := 8, 	fn := 1),            	// 1 Hodnota minimum
            (wh:=13, x:= 50   ,y:= y1 + 250, w:= x2-110, h :=251,		FgC := 4, BgC := 6, 	fn := 2),              	// 2 Hodnota maximum
				(wh:=221,x:= 50	,y:= y1 + 320, w:= 25 , 	h := 30, 	FgC := 4, BgC := 5, 	fn :=149),              // 3 hodnota 0..100%

            (wh:=13, x:= 50   ,y:= y1 + 440, w:= x2-110, h :=251,		FgC := 4, BgC := 3, 	fn := 0),            	// 4 Korekcia - Konverzý faktor
            (wh:=221,x:= 50	,y:= y1 + 480, w:= 25 , 	h := 33,  	FgC :=4,  BgC := 3, 	fn :=120,),          	// 5 hodnota po korekcii

				(wh:=13, x:= 50   ,y:= y1 + 600, w:= x2-110 ,h :=251,		FgC := 4, BgC := 2, 	fn := 3),              	// 6 povolena zmena
            (wh:=13, x:= 50   ,y:= y1 + 680, w:= x2-110 ,h :=251,		FgC := 4, BgC := 2, 	fn := 4),              	// 7 opozdnie zmeny
            (wh:=13, x:= 50   ,y:= y1 + 760, w:= x2-110 ,h :=251,  	FgC := 4, BgC := 2, 	fn := 5),              	// 8 opozdnie zmeny
			   (wh:=20, x:=x2-60 ,y:= y1 + 820, w:= 48     , 				FgC := 0, BgC :=50, 	fn := 241),	  				// 9 neposielat do room
			   (wh:=20, x:=x2-60 ,y:= y1 + 880, w:= 48     , 				FgC := 4, BgC :=50, 	fn := 100)  				//10 zablokovat
       )];

      s  : ARRAY[0..5] OF NH_SLD_DAT := [
            ( t:=0, xv := x2-53, v1:=1.0, 	v2 := 200.0,  fmt := '%5.1f',   	txt:= 148, ink:=0.1),      	// 0 Korekcia - Konverzý faktor
            ( t:=0, xv := x2-53, v1:=-40.0, 	v2 := 1000.0, fmt := '%5.0f',   	txt:= 130),      					// 1 Hodnota minimum
            ( t:=0, xv := x2-53, v1:=-40.0, 	v2 := 1000.0, fmt := '%5.0f',   	txt:= 131),      					// 2 Hodnota maximum
            ( t:=0, xv := x2-53, v1:=0.0, 	v2 := 10.0 ,  fmt := '%5.1f', 	txt:= 121, ink:=0.1),			// 3 povolena zmena
            ( t:=1, xv := x2-53, v1:=0.0, 	v2 := 254.0 , fmt := '%5.0f',   	txt:= 122),       				// 4 opozdenie zmeny
            ( t:=3, xv := x2-53, v1:=0.0, 	v2 := 3599.0, fmt := 's%Tmm:ss m', 	txt:= 609)       			// 5 odoberat vzorky
			];

   END_STRUCT;
   NH_FRM_059 {HIDDEN}  :  STRUCT
      hed      : NH_FRM_HED := (Name:='_059',wht:=3);
      mnu      : NH_MNU := ( n:=3,                                  				// MNU-GATE
                        o := [
                              (fn :=   6,wh:=  6,cm :=  31),
                              (),
                              (fn :=  83,wh:= 84,cm := 205,x:=xc-90 ,frm:=58),       	// nastavenia
										(fn := 348,wh:=348,cm :=  82,x:=xc   			),				// ROM->DEV
                              (fn :=330,wh:=330,cm := 205,x:=xc+90   ,frm:=60)       	// HW-parametre

                           ]);
   END_STRUCT;

   NH_FRM_060  {HIDDEN} : STRUCT      // HW - typ premennej
      hed      : NH_FRM_HED := (Name:='_060',wht:=2,row:=1,sld:=0);
      mnu   : NH_OBJ_123 := // 2 riadky
            (wh:=123,cf:=(x:= xc-40,     y:= y1 + 80, typ:=1, rw2:=7, h:= 50, hTxt:= 28),
                 txt:=[482,483,484,485,486,487,488]);                                                    // 1 rolovaci vyber textov
      ROW   : ARRAY[2..10] OF NH_OBJ_DAT ;
   END_STRUCT

   NH_FRM_061  {HIDDEN} :  STRUCT 	// FRM - setup SVD,SVA,ZAS,SIR
      hed      : NH_FRM_HED := (Name:='_061',wht:=2,row:=1,sld:=6);
      mnu   : NH_OBJ_123 := // 2 riadky
            (wh:=123,cf:=(x:= xc-150,     y:= y1 + 80, typ:=1, rw2:=6, h:= 50, hTxt:= 28),
                 txt:=[490,491,492,493,494,495]);                                                    // 1 rolovaci vyber textov
      ROW   : ARRAY[2..10] OF NH_OBJ_DAT := [
				(),
				(),
				(),
				(),
				(),
            (wh:=20, x:= x2-140  , y:= y1 + 700,   w:= 48     , FgC := 0, BgC :=50          , fn := 146          ), // 7 obnovit po restarte
            (wh:=20, x:= x2-140  , y:= y1 + 760,   w:= 48     , FgC := 0, BgC :=50          , fn := 506          ), // 8 RGBWA
            (wh:=20, x:= x2-140  , y:= y1 + 820,   w:= 48     , FgC := 0, BgC :=50          , fn := 228          ),  // 9 archivovat
            (wh:=20, x:= x2-140  , y:= y1 + 880,   w:= 48     , FgC := 4, BgC :=50          , fn := 100          ) //10 zablokovat

             ];

      s  : ARRAY[0..5] OF NH_SLD_DAT :=
           [
            (t := 0,      		v2:= 3000.0 , fmt := '%4.0f W'            , txt:=  69),        // 0 Prikon
            (t := 1                       , fmt := '%3.0f %%'       		, txt:=  70),      	// 1 stmievatelne minimum
            (t := 1                       , fmt := '%3.0f %%'       		, txt:=  71),       	// 2 efektivma maximum
            (t := 1, v1:=1.0, v2:=10      , fmt := '%3.0f'        		, txt:= 365),       	// 3 krok stmievania Fade Rate
            (t := 1, v1:=1.0, v2:=10      , fmt := '%3.0f'         		, txt:= 364),       	// 4 Fade Time
            (t := 1,          v2:=50.0 	, fmt := '1%Ts.z s'           , txt:= 145)        	// 5 opozdene zazati  po vypnuti
              ];
   END_STRUCT;

   NH_FRM_062 {HIDDEN}:  STRUCT 	//39 FRM - LED WSB/TGL
      hed      : NH_FRM_HED := (Name:='_062',wht:=2,row:=1,sld:=8);
      r  : ARRAY[1..2] OF NH_ROW_O := [( ob := [
            (wh:=13, x:= 50     , y:= y1 + 100,   w:= x2-110  ,FgC := 4, BgC := 7,h:=250   , fn := 0             ), // Den-intensita
            (wh:=13, x:= 50     , y:= y1 + 200,   w:= x2-110  ,FgC := 4, BgC := 8,h:=250   , fn := 1             ), // 253 znamena, ze zmenu slidera bude ukladat do nejakej BOOL premennej
            (wh:=13, x:= 50     , y:= y1 + 300,   w:= x2-110  ,FgC := 4, BgC := 9,h:=250   , fn := 2             ),
            (wh:=13, x:= 50     , y:= y1 + 400,   w:= x2-110  ,FgC := 4, BgC := 4,h:=250   , fn := 3             ),
            (wh:=13, x:= 50     , y:= y1 + 500,   w:= x2-110  ,FgC := 4, BgC :=30,h:=250   , fn := 4             ), // Den-cas uspatia
            (wh:= 0, x:= 50     , y:= y1 + 550,   w:= x2-110  ,FgC := 4, BgC := 3,h:=250   , fn := 5             ),
            (wh:= 0, x:= 50     , y:= y1 + 630,   w:= x2-110  ,FgC := 4, BgC := 9,h:=250   , fn := 6             ),
            (wh:= 0, x:= 50     , y:= y1 + 710,   w:= x2-110  ,FgC := 4, BgC := 3,h:=250   , fn := 7             ),
//            (wh:= 0, x:= x2/2   , y:= y1 + 380,   w:= 400    , FgC := 2, fn := 2, h:=25, cf:=(n:=139),nTch:=1    ),  // 'Uspat po case'
            (wh:= 0, x:= x2-60  , y:= y1 + 770,   w:= 48, Fn :=480,  FgC :=10, BgC := 50, h := 0, cf :=(c:=3), cm:=140  ),  // 8 LED nad funcnym tlacitkom
            (wh:= 0, x:= x2-60  , y:= y1 + 830,   w:= 48     , FgC := 0, BgC :=50          , fn := 55            ),  // 9  pohyb resetuje cas
            (wh:= 0, x:= x2-60  , y:= y1 + 880,   w:= 48     , FgC := 0, BgC :=50          , fn := 111           )   //10  zobudit pohybom
              ]), ( ob := [
            (wh:= 0, x:= x2/2   , y:= y1 +  40,   w:= 400    , FgC := 2, fn := 2, h:=25, cf:=(n:=137),nTch:=1    ),   // 'Svietivost'
            (wh:= 0, x:= x2/2   , y:= y1 + 410,   w:= 400    , FgC := 2, fn := 2, h:=25, cf:=(n:=139),nTch:=1    )  // 'Uspat po case'
              )];
      s  : ARRAY[0..7] OF NH_SLD_DAT :=
           [
            (t := 1, v2:=254,       fmt := '%3.0f '            , txt:= 500),        // 0 Den - intenzita
            (t := 1, v2:=254,       fmt := '%3.0f '            , txt:= 501),        // 1 Vecr
            (t := 1, v2:=254,       fmt := '%3.0f '            , txt:= 502),        // 2 Noc
            (t := 1, v2:=254,       fmt := '%3.0f '            , txt:= 503),        // 3 Rano
            (t := 1, v2:=254,       fmt := '%3.0f '            , txt:= 504)         // 4 Rano
              ];

   END_STRUCT;
   NH_FRM_063 {HIDDEN}  :  STRUCT
      hed      : NH_FRM_HED := (Name:='_063',wht:=3);
      mnu      : NH_MNU := ( n:=3,                                  				// MNU-ROL - hlavneme menu
                        o := [
                              (fn :=   6,wh:=  6,cm :=  31),
                              (),
                              (fn :=  85,wh:= 85,cm := 205, frm:=82),    						// nastavit roletu
                              (fn := 261,wh:=262,cm := 205, frm:=67), 	// vietor
                              (fn := 130,wh:=131,cm := 205, frm:=66),   // sumrak
                              (fn := 139,wh:=140,cm := 205),        		// Slnko
										(),
                              (fn :=  23,wh:= 24,cm := 203, frm:=81)    // setup - odskoci sadodalsieho menu o uroven dalej
                           ]);
   END_STRUCT;

   NH_FRM_064 {HIDDEN}:  STRUCT 	// FRM-ROL lvl
      hed      : NH_FRM_HED := (Name:='_064',wht:=2,row:=1,sld:=9);
      r  : ARRAY[1..1] OF NH_ROW_O := [( ob := [
//            (wh:=0, x:= 50     , y:= y1 + 150,   w:= x2-110  ,FgC := 4, BgC := 9          , fn := 0             ), // 0 Rolete
			   (wh:=20, x:=x2-60  , y:= y1 +  60,   w:= 48     , 				FgC := 0, BgC :=50, fn := 607),	  		// 9 neposielat do room
            (wh:=0,  x:= 50    , y:= y1 + 230,   w:= x2-110  ,FgC := 4, BgC := 2          , fn := 1             ), // 1 Lamela
            (wh:=0,  x:= 50    , y:= y1 + 310,   w:= x2-110  ,FgC := 4, BgC := 5          , fn := 6             ), // 2 s opozdenim
            (wh:=6,  x:= x2/2  , y:= y1 + 150,   w:= 400    , FgC := 3, BgC := 0, fn := 2, h:=30,cf:=(n:=114)   ), // 3 text Predvolby
            (wh:=13, x:= 50    , y:= y1 + 250,   w:= x2-110  ,FgC := 4, BgC := 2          , fn := 2             ), // 4 pv1
            (wh:=13, x:= 50    , y:= y1 + 330,   w:= x2-110  ,FgC := 4, BgC := 2          , fn := 3             ), // 5 pv2
            (wh:=13, x:= 50    , y:= y1 + 410,   w:= x2-110  ,FgC := 4, BgC := 2          , fn := 4             ), // 6 pv3
            (wh:=13, x:= 50    , y:= y1 + 480,   w:= x2-110  ,FgC := 4, BgC := 2          , fn := 5             ), // 7 pv4
            (wh:=13, x:= 50    , y:= y1 + 830,   w:= x2-110  ,FgC := 4, BgC := 3          , fn := 7             ), // 8 pauza medzi predvolbami
            (wh:=13, x:= 50    , y:= y1 + 700,   w:= x2-110  ,FgC := 4, BgC := 3          , fn := 8             ), // 9 typ
            (wh:=0, x:= x2-60  , y:= y1 +  50,   w:= 48     , FgC := 0, BgC :=50          , fn := 246           ) //10 nastavit predvolenu poziciu
//            (wh:= 6, x:=xc      , y:= 1015,       w:= 400, h:=20, Fgc:=2, fn:=2, nTch:=1, cf:=(c:=254)           )  // 10 info dali nbr {len admin}
              )];
      s  : ARRAY[0..8] OF NH_SLD_DAT :=
           [
            (t := 1, v2:=100,       fmt := '%3.0f %%'            , txt:= 112),        // 0 Rol
            (t := 1, v2:=100,       fmt := '%3.0f %%'            , txt:= 113),        // 1 LAm
            (t := 1, v2:=100,       fmt := '%3.0f %%'            , txt:=   0),        // 2 pv1
            (t := 1, v2:=100,       fmt := '%3.0f %%'            , txt:=   0),        // 3 pv2
            (t := 1, v2:=100,       fmt := '%3.0f %%'            , txt:=   0),        // 4 pv3
            (t := 1, v2:=100,       fmt := '%3.0f %%'            , txt:=   0),        // 5 pv4
            (t := 3, v2:=1800,      fmt := 's%Tm:ss m'           , txt:= 115),        // 6 opozdenie
            (t := 1, v2:=180,       fmt := '%3.0f°'              , txt:= 251),         // 7 typ uhla lamely
            (t := 1, v2:=15,        fmt := '1%Ts.z s'            , txt:= 239) // 8 pauza medzi predvolbami
              ];
   END_STRUCT;

   NH_FRM_065 {HIDDEN}:  STRUCT 	// FRM-ROL Up/dn
      hed      : NH_FRM_HED := (Name:='_065',wht:=2,row:=1,sld:=10);
      r  : ARRAY[1..1] OF NH_ROW_O := [( ob := [
//            (wh:=6,  x:= x2/2    , y:= y1 + 50,    w:= 400    , FgC := 3, BgC := 0, fn := 2, h:=30,cf:=(n:=194)   ), // 0 text Pohyb hore
            (wh:=13, x:= 50     , y:= y1 +  80,   w:= x2-110  ,FgC := 4, BgC := 3          , fn := 0             ), // 0 Cas vytiahnutia
            (wh:=13, x:= 50     , y:= y1 + 160,   w:= x2-110  ,FgC := 4, BgC := 3          , fn := 1             ), // 1 otvorenia
            (wh:=13, x:= 50     , y:= y1 + 240,   w:= x2-110  ,FgC := 4, BgC := 3          , fn := 2             ), // 2 Opozdenie motora On/Off
            (wh:=13, x:= 50     , y:= y1 + 340,   w:= x2-110  ,FgC := 4, BgC := 3          , fn := 8             ), // 3 Opozdenie motora zmena smeru

				(wh:=13, x:= 50     , y:= y1 + 460,   w:= x2-110  ,FgC := 4, BgC := 5          , fn := 3             ), // 4 zatiahnutie
            (wh:=13, x:= 50     , y:= y1 + 540,   w:= x2-110  ,FgC := 4, BgC := 5          , fn := 4             ), // 5 zaklopenie
            (wh:=13, x:= 50     , y:= y1 + 620,   w:= x2-110  ,FgC := 4, BgC := 5          , fn := 5             ), // 6 opozdenie motora
            (wh:=13, x:= 50     , y:= y1 + 700,   w:= x2-110  ,FgC := 4, BgC := 5          , fn := 9             ), // 7 opozdenie motora zmena smeru

            (wh:=13, x:= 50     , y:= y1 + 820,   w:= x2-110  ,FgC := 3, BgC :=4          , fn := 6             ), // 8 ochranna doba - reverzia
            (wh:=13, x:= 50     , y:= y1 + 900,   w:= x2-110  ,FgC := 3, BgC :=4          , fn := 7             ), // 9 predlzit dojazd
            (wh:= 0, x:= x2-60  , y:= y1 + 830,   w:= 48     , FgC := 0, BgC :=50          , fn := 55            )  // 10
              )];
      s  : ARRAY[0..9] OF NH_SLD_DAT :=
           [
            (t := 3, v1:=500,v2:=12000,      fmt := '2%Tm:ss.z m'         	, txt:= 196, ink:=10.0),   // 0 Up Rol
            (t := 3, 			v2:=4000,     	fmt := '0%Ts.zz s'        		, txt:= 198, ink:=10.0),   // 1 Up Lam
            (t := 1, 			v2:=100,       fmt := '2%Ts.zz s'          	, txt:= 192, ink:=1.0),   // 2 Up Mot
            (t := 3, v1:=500,v2:=12000,      fmt := '2%Tm:ss.z m'         	, txt:= 197, ink:=10.0),   // 3 Dn Rol
            (t := 3, 			v2:=4000,      fmt := '0%Ts.zz s'      			, txt:= 199, ink:=10.0),   // 4 Dn Lam
            (t := 1, 			v2:=100,       fmt := '2%Ts.zz s'          	, txt:= 192, ink:=1.0),   		// 5 UpMot
            (t := 1, 			v2:=50, v1:=5, fmt := '1%Ts.z s'            	, txt:=  98),         			// 6 ochranna doba
            (t := 1, 			v2:=10,        fmt := 's%Ts s'          	   , txt:= 191),   					// 7 Predlzit dojazd
            (t := 1, 			v2:=100,       fmt := '2%Ts.zz s'          	, txt:= 240),   					//  8 opozdenie up - zmena smeru
            (t := 1, 			v2:=100,       fmt := '2%Ts.zz s'          	, txt:= 240)   					//  9 opozdenie Dn - zmena smeru
              ];
   END_STRUCT;

   NH_FRM_066 {HIDDEN}:  STRUCT 	// FRM-ROL SUMRAK
      hed      : NH_FRM_HED := (Name:='_066',wht:=2,row:=1,sld:=8);
      r  : ARRAY[1..1] OF NH_ROW_O := [( ob := [
            (wh:=20, x:= x2-60  , y:= y1 +  50,   w:= 48     , FgC := 0, BgC :=50          , fn := 249           ), // 0 ovplyvnuje sumrak v miestnosti
            (wh:=13, x:= 50     , y:= y1 + 150,   w:= x2-110  ,FgC := 4, BgC := 3   		  , fn := 0             ), // 1 Rolete
            (wh:=13, x:= 50     , y:= y1 + 250,   w:= x2-110  ,FgC := 4, BgC := 3   		  , fn := 1             ), // 2 Lamela
            (wh:=13, x:= 50     , y:= y1 + 350,   w:= x2-110  ,FgC := 4, BgC := 5   		  , fn := 2             ), // 3 podiel na dark
            (wh:= 0, x:= x2/2    , y:= y1 + 370,   w:= 400    , FgC := 3, BgC := 0, fn := 2, h:=30,cf:=(n:=114)   ), // 4 text Predvolby
            (wh:= 0, x:= 50     , y:= y1 + 460,   w:= x2-110  ,FgC := 4, BgC := 2          , fn := 2             ), // 5 pv1
            (wh:= 0, x:= 50     , y:= y1 + 540,   w:= x2-110  ,FgC := 4, BgC := 2          , fn := 3             ), // 6 pv2
            (wh:= 0, x:= 50     , y:= y1 + 620,   w:= x2-110  ,FgC := 4, BgC := 2          , fn := 4             ), // 7 pv3
            (wh:= 0, x:= 50     , y:= y1 + 700,   w:= x2-110  ,FgC := 4, BgC := 2          , fn := 5             ), // 8 pv4
            (wh:= 0, x:= x2-60  , y:= y1 +  50,   w:= 48     , FgC := 0, BgC :=50          , fn := 249           ), //
            (wh:=20, x:= x2-60  , y:= y1 + 800,   w:= 48     , FgC := 0, BgC :=50          , fn := 250           )  // Naklapanie lamiel HW
              )];

      s  : ARRAY[0..7] OF NH_SLD_DAT :=
           [
            (t := 1, v2:=100,       fmt := '%3.0f %%'            , txt:= 248),        // 0 Rol
            (t := 1, v2:=100,       fmt := '%3.0f %%'            , txt:= 247),        // 1 LAm
            (t := 1, v2:=100,       fmt := '%3.0f %%'            , txt:= 245),        // 2 podiel na Dark
            (t := 1, v2:=100,       fmt := '%3.0f %%'            , txt:=   0),        // 3 pv2
            (t := 1, v2:=100,       fmt := '%3.0f %%'            , txt:=   0),        // 4 pv3
            (t := 1, v2:=100,       fmt := '%3.0f %%'            , txt:=   0),        // 5 pv4
            (t := 3, v2:=1800,      fmt := 's%Tm:ss m'           , txt:= 115),        // 6 opozdenie
            (t := 1, v2:=180,       fmt := '%3.0f°'              , txt:= 251)         // 7 typ uhla lamely
              ];
   END_STRUCT;

   NH_FRM_067 {HIDDEN}:  STRUCT 	// FRM-ROL WIND
      hed      : NH_FRM_HED := (Name:='_067',wht:=2,row:=1,sld:=8);
      r  : ARRAY[1..1] OF NH_ROW_O := [( ob := [
            (wh:=20, x:= x2-60  ,y:= y1 +  50,   w:= 48     , FgC := 0, BgC :=50          , fn := 525           	), // 0 povolit ochranu pred vetrom
            (wh:=13, x:= 50     ,y:= y1 + 150,   w:= x2-110  ,FgC := 4, BgC :=17   		  , fn := 0             	), // 1 Silny vietor je >
            (wh:=13, x:= 50     ,y:= y1 + 230,   w:= x2-110  ,FgC := 4, BgC :=17   		  , fn := 1             	), // 2 vytiahnut po case
            (wh:=13, x:= 50     ,y:= y1 + 330,   w:= x2-110  ,FgC := 4, BgC := 8          , fn := 2             	), // 3 vratit spat po case
            (wh:=13, x:= 50     ,y:= y1 + 420,   w:= x2-110  ,FgC := 4, BgC := 8          , fn := 3             	), // 4 ak je vietor menasi ako
            (wh:=6,  x:= xc    , y:= y1 + 490,   w:= 400    , FgC := 4, BgC := 0, fn := 2, h:=28,cf:=(n:=530)   	), // 5 odlozit vratenie daymode
            (wh:=20, x:= 80  , 	y:= y1 + 540,   w:= 48, Fn :=0,  FgC :=1, BgC := 50, w:=62, h := 110, cf :=(c:=4)),	// 6 Daymode
            (wh:=20, x:= x2-60  ,y:= y1 + 610,   w:= 48     , FgC := 0, BgC :=50          , fn := 242           	), // 7 len ked fuka vietor >
            (wh:=13, x:= 50     ,y:= y1 + 710,   w:= x2-110  ,FgC := 4, BgC := 3          , fn := 4             	), // 8 smer od
            (wh:=13, x:= 50     ,y:= y1 + 790,   w:= x2-110  ,FgC := 4, BgC := 3          , fn := 5             	), // 9 smer do
            (wh:=13, x:= 50     ,y:= y1 + 900,   w:= x2-110  ,FgC := 4, BgC := 17          , fn := 6             	) //10 zablokovat rucnym zasah
              )];
      s  : ARRAY[0..7] OF NH_SLD_DAT :=
           [
            (t := 1, v2:=25,    v1:=1.0,  fmt := '%2.0f m/s'           	, txt:= 526),         // 0 silny vietor
            (t := 1, v2:=255,   v1:=1.0,  fmt := 's%Tm:ss m'           	, txt:= 527),        // 1 po akom case sa vytiahnu
            (t := 1, v2:=120,   v1:=1.0,  fmt := 'm%Th:mm h'           	, txt:= 528),        // 2 po akom èase sa vrátia
            (t := 1, v2:=25,        		fmt := '%2.0f m/s'            , txt:= 529),         // 3 ked vietor poklesne
            (t := 3, v2:=360,       		fmt := '%3.0f °'            	, txt:= 243),        // 4 WinDirFrom
            (t := 3, v2:=360,       		fmt := '%3.0f °'            	, txt:= 244),        // 5 WinDirTo
            (t := 3, v2:=360,       		fmt := 'm%Th:mm h'           	, txt:= 356),        // 6 rucny zasah blokuje
            (t := 1, v2:=180,       		fmt := '%3.0f°'              	, txt:= 251)         // 7 typ uhla lamely
              ];
   END_STRUCT;
   NH_FRM_068 {HIDDEN}  :  STRUCT
      hed      : NH_FRM_HED := (Name:='_068',wht:=3);
      mnu      : NH_MNU := ( n:=3,                                  				// MNU-GATE
                        o := [
                              (fn :=   6,wh:=  6,cm :=  31),
                              (fn := 385,wh:=385,cm := 0),
										(fn := 385,wh:=385,cm := 205,x:=xc-90, frm:=69),		// meteostanica
                              (fn := 261,wh:=262,cm := 205,x:=xc, 	frm:=80),    	// wind
                              (fn :=  23,wh:= 24,cm := 205,x:=xc+90, frm:=84)    	// setup
									]);
   END_STRUCT;

   NH_FRM_069 {HIDDEN}:  STRUCT 	// FRM-ROL lvl
      hed      : NH_FRM_HED := (Name:='_069',wht:=2,row:=1,sld:=0);
      r  : ARRAY[0..7] OF NH_OBJ_DSH := [
				(x:=xc-140,	y:=y1+180,	w:=280,	dash:=380, vMin:=  0.0, vMax:=  20.0,tx1:= 'Avg', title:=513, idx:=0, mj:='m/s'),	// rychost vetra
				(x:=xc+150,	y:=y1+180,	w:=280,	dash:=381, vMin:=860.0, vMax:=1090.0,tx1:= 'Min',title:=514,  idx:=1, mj:='hPa'),	// atmosfericky tlak

				(x:=xc-140,	y:=y1+400,	w:=280,	dash:=382, vMin:=-10.0, vMax:=  40.0,tx1:= 'Min', title:=515, idx:=2, mj:='°C'),		// teplota
				(x:=xc+150,	y:=y1+400,	w:=280,	dash:=382, vMin:=-10.0, vMax:=  40.0,tx1:= 'Min', title:=516, idx:=3, mj:='°C'),		// winchill - pocit.teplota

				(x:=xc-140,	y:=y1+620,	w:=280,	dash:=381, vMin:= 0.0,  vMax:= 100.0,tx1:= 'Min', title:=517, idx:=4, mj:='%'),		// relativna vlhost
				(x:=xc+150,	y:=y1+620,	w:=280,	dash:=381, vMin:= 0.0,  vMax:= 100.0,tx1:= 'Min', title:=518, idx:=5, mj:='g/m'),	// absolutna vlkost

				(x:=xc-140,	y:=y1+840,	w:=280,	dash:=380, vMin:= 0.0,  vMax:=1400.0,tx1:= 'Min', title:=519, idx:=6, mj:='W/m'),	// sl.ziarenie
				(x:=xc+150,	y:=y1+840,	w:=280,	dash:=383, vMin:= 0.0,  vMax:= 100.0,tx1:= 'Min', title:=520, idx:=7, mj:='km')		// burka
				];
      o  : ARRAY[8..10] OF NH_OBJ_DAT := [
            (wh:=101,  x:= xc        , y:= y1 + 65 ,   w:= 75     , Fgc :=3 , BgC := 3, btn:=1),       // 1 smer prudenia
            (wh:=0)    // 3 text Predvolby
              ];
   END_STRUCT;

   NH_FRM_070  {HIDDEN} : STRUCT      // ventil vody
      hed      : NH_FRM_HED := (Name:='_070',wht:=2,row:=1,sld:=1);
      mnu   : NH_OBJ_123 := // 2 riadky
            (wh:=123,cf:=(x:= xc-200,     y:= y1 + 100, typ:=1, rw2:=3, h:= 50, hTxt:= 28),
                 txt:=[521,522,523]);                                                    // 1 rolovaci vyber textov
      ROW   : ARRAY[2..10] OF NH_OBJ_DAT := [
             (wh:=13, x:= 50     , y:= y1 + 600,   w:= x2-110  ,FgC := 4, BgC := 3   		   , fn := 0   ), //2 Lamela
             (wh:=20, x:= x2-60  , y:= y1 + 700,   w:= 48     , FgC := 0, BgC :=50          , fn := 146 ), // 3 obnovit stav po restarte
             (wh:=20, x:= x2-60  , y:= y1 + 800,   w:= 48     , FgC := 4, BgC :=50			  	, fn := 100	) // 8 zablokovat
					];
      s  : ARRAY[0..0] OF NH_SLD_DAT :=
           [
            (t := 1, v2:=60,       fmt := '%3.0f s'            , txt:= 116)        // 0 Rol
              ];
   END_STRUCT
   NH_FRM_071 {HIDDEN}  :  STRUCT
      hed      : NH_FRM_HED := (Name:='_071',wht:=3);
      mnu      : NH_MNU := ( n:=1,
                        o := [
                              (fn :=   6,wh:=  6,cm :=  31),
                              (),
                              (fn := 120,wh:=121,cm := 205, frm:=72),      // cas
                              (fn := 149,wh:=149,cm := 205, frm:=72),      // SunSet/Sunrise
                              (fn := 130,wh:=131,cm := 205, frm:=72),      // Dark/Light
                              (fn := 387,wh:=387,cm := 205, frm:=74),      // RND
//		                        (fn:= 23,wh:= 24,cm := 205, frm:=74),    		// setup
										(fn:=  0),
										(fn:=348,wh:=348,cm :=  82   			)		  	// ROM->DEV
                           ]);
   END_STRUCT;

   NH_DAYS_OF_WEEK  {HIDDEN}  : STRUCT      	// typove dni + PO-NE
      txt   : ARRAY[0..10] OF NH_OBJ_DAT :=
          [ (wh:=105,x:=70,  y:=y1+805, w:= 64,h:=64,FgC:=3,BgC:=4,cf:=(n:=201)),  		// 0 -> 1 PO Fgc=kruh,BgC:=text
			 	(wh:=105,x:=145,  			 w:= 64,h:=64,FgC:=3,BgC:=4,cf:=(n:=201)),  		// 1 -> 2 UT
			 	(wh:=105,x:=220,            w:= 64,h:=64,FgC:=3,BgC:=4,cf:=(n:=201)),   	// 2 -> 3 ST
			 	(wh:=105,x:=295,            w:= 64,h:=64,FgC:=3,BgC:=4,cf:=(n:=201)),   	// 3 -> 4 ST
			 	(wh:=105,x:=370,            w:= 64,h:=64,FgC:=3,BgC:=4,cf:=(n:=201)),   	// 4 -> 5 PI
			 	(wh:=105,x:=445,            w:= 64,h:=64,FgC:=3,BgC:=4,cf:=(n:=201)),   	// 5 -> 6 SO
			 	(wh:=105,x:=520,            w:= 64,h:=64,FgC:=3,BgC:=4,cf:=(n:=201)),   	// 6 -> 7 NE

			 	(wh:=105,x:= 70,            w:= 64,h:=64,FgC:=3,BgC:=4,cf:=(n:=202),fn:=273),   	// 7 -> 8 sviatok
			 	(wh:=105,x:=145,            w:= 64,h:=64,FgC:=3,BgC:=4,cf:=(n:=203),fn:=276),   	// 8 -> 9 party
			 	(wh:=105,x:=220,            w:= 64,h:=64,FgC:=3,BgC:=4,cf:=(n:=204),fn:=279),   	// 9 -> 10 sviatok
			 	(wh:=105,x:=295,            w:= 64,h:=64,FgC:=3,BgC:=4,cf:=(n:=205),fn:=282)   	//10 -> 11 party
			];

   END_STRUCT

   NH_FRM_072 {HIDDEN}:  STRUCT 	// FRM-TIM  0=Nacasovat,1=cyklus,2=Sunrise,3=Sunshine,4=Dark,5=Light
      hed      : NH_FRM_HED := (Name:='_072',wht:=2,row:=4,sld:=6);
      r1o0_1_Type : NH_OBJ_123 :=                     // 2 objekty
      	(	wh:=123,cf:=(x:= xc-220,     y:= y1 + 50, typ:=1, rw1:=1, rw2:=2, h:= 40, hTxt:= 28),
            txt:=[542,543,544,545,546,547]
			);
      r1o2_3_OnOff : NH_OBJ_123 := // On/Off/On+Off
      	(	wh:=123,cf:=(x:= xc-140,     y:= y1 + 150, typ:=1, rw2:=3, h:= 45, hTxt:= 28),
            txt:=[539,540,541]
			);
      r1o4_10  	: ARRAY[4..10] OF NH_OBJ_DAT :=
			[
            (wh:=13, x:=50    , y:= y1+ 540,w:= x2-110  ,FgC := 4, BgC := 5 , fn := 2 ), 	//2 Cas vypnutia
            (wh:=13, x:=50    , y:= y1+ 620,w:= x2-110  ,FgC := 4, BgC := 6 , fn := 3 ), 	//3 Cas zapnutia
				(wh:=0),
				(wh:=0),
				(wh:=0),
			 	(wh:=20, x:=70   , y:= y1+ 890,FgC :=13, w:=74, h := 72, cf :=(c:=3)), 			//9 Lock/Dark
			  	(wh:=20, x:=369  , y:= y1+ 730,FgC :=12, w:=48, h := 49, cf :=(c:=3))	];			//10 Daymode

		r2		: NH_DAYS_OF_WEEK;
		r3_On	: NH_DAT_TIM2:= ( txt := [          // riadok 3
						(fn:=0,FgC:=0,nTch:=1,y:=y1+320),							// fn:=0 ... hlavny {1.riadok}
						(wh:=0),
						(wh:=0),
						(wh:=0),
	      	      (wh:=125,x:=xc+130,w:= 28,h:=28,FgC:=4),          	// 4 hour
   	      	   (wh:=125,x:=xc+190,w:= 28,h:=28,FgC:=5),          	// 5 min
      	      	(wh:=  0,x:=xc+250,w:= 28,h:=28,FgC:=6),          	// 6 sec
						(wh:=0),
	   	         (wh:=0), 																			// 8 text v urovni navestie
   	   	      (wh:=125, x:=50,w:=200,FgC:=10,BgC:=0, fn:=0, h:=28,cf:=(n:=82), nTch:=1), // 9 text vacsinou pred datumom
	   	   	   (wh:=13,x:=50, y:=y1+450, w:=x2-110 ,FgC:=4, BgC:=3, fn:=1)
						]);

		r4_Off	: NH_DAT_TIM2 := ( txt := [            // riadok 4 ToDate
						(fn:=3,FgC:=0,nTch:=1,y:=y1+360),							// fn:=0 ... hlavny {1.riadok}
						(wh:=0),
						(wh:=0),
						(wh:=0),
	      	      (wh:=125,x:=xc+130,	w:= 28,h:=28,FgC:=4),          	// 4 hour
   	      	   (wh:=125,x:=xc+190, 	w:= 28,h:=28,FgC:=5),          	// 5 min
      	      	(wh:=  0,x:=xc+250,	w:= 28,h:=28,FgC:=6),          	// 6 sec
						(wh:=0),
	   	         (wh:=0), // text v urovni navestie
   	   	      (wh:=125, x:=50, y:=y1+450, 		w:=200,FgC:=10,BgC:=0, fn:=0, h:=28,cf:=(n:=83), nTch:=1), // text vacsinou pred datumom
	   	   	   (wh:=0)
						]);

      s  : ARRAY[0..5] OF NH_SLD_DAT :=
         [  (t:=1,v1:=1, v2:=31, fmt := '%3.0f', txt:= 116, zom:=0,tun:=0),        	// 0 slider k start
				(t:=1,v1:=0, v2:=59, fmt := '%3.0f', txt:= 116, zom:=0,tun:=0),        	// 1 slider k Stop
            (t:=3, v2:=300,      fmt := 'm%Th:mm h'           , txt:= 551),			// 2 cas vypnutia
            (t:=3, v2:=300,      fmt := 'm%Th:mm h'           , txt:= 552)          // 3 cas zapnutia
         ];
   END_STRUCT;

   NH_FRM_073 {HIDDEN}:  STRUCT 	// FRM-TIM  Nacasovat/cyklus  Sunrise/Sunshine, Datk/Light
      hed      : NH_FRM_HED := (Name:='_073',wht:=2,row:=2,sld:=6);
      r1o0_1_Type : NH_OBJ_123 :=                     // 2 objekty
      	(	wh:=123,cf:=(x:= xc-220,     y:= y1 + 50, typ:=1, rw1:=3, rw2:=4, h:= 40, hTxt:= 28),
            txt:=[542,543,544,545,546,547]       	// Typ casovaca
			);
      r1o2_3_OnOff : NH_OBJ_123 := // On/Off/On+Off
      	(	wh:=123,cf:=(x:= xc-140,     y:= y1 + 260, typ:=1, rw2:=3, h:= 45, hTxt:= 28),
            txt:=[539,540,541]
			);
      r1o4_10  	: ARRAY[4..10] OF NH_OBJ_DAT :=
			[
            (wh:=13, x:=50    , y:= y1+ 540,w:= x2-110  ,FgC := 4, BgC := 5 , fn := 2 ), 	//4 Vykonat oneskorene
            (wh:=13, x:=50    , y:= y1+ 620,w:= x2-110  ,FgC := 4, BgC := 6 , fn := 3 ), 	//5 Vypnut po case
				(wh:=0),
				(wh:=0),
				(wh:=0),
			 	(wh:=20, x:=70   , y:= y1+ 890,FgC :=13, w:=74, h := 72, cf :=(c:=3)), 			//9 Lock/Dark
			  	(wh:=20, x:=369  , y:= y1+ 730,FgC :=12, w:=48, h := 49, cf :=(c:=3))	];			//10 Daymode

		r2		: NH_DAYS_OF_WEEK;

      s  : ARRAY[0..5] OF NH_SLD_DAT :=
         [  (t:=1,v1:=1, v2:=31, fmt := '%3.0f', txt:= 116, zom:=0,tun:=0),        	// 0 slider k start
				(t:=1,v1:=0, v2:=59, fmt := '%3.0f', txt:= 116, zom:=0,tun:=0),        	// 1 slider k Stop
            (t:=3, v2:=600,      fmt := 'm%Th:mm h'           , txt:= 115),			// 4 vykonat oneskorene
            (t:=3, v2:=600,      fmt := 'm%Th:mm h'           , txt:=  64)          // 5 vypnut po case
         ];
   END_STRUCT;

   NH_FRM_074 {HIDDEN}:  STRUCT 	// FRM-TIM  len typ:=6: Random
      hed      : NH_FRM_HED := (Name:='_074',wht:=2,row:=2,sld:=7);
      r1o0_1_Type : NH_OBJ_123 :=                     // 2 objekty
      	(	wh:=123,cf:=(x:= xc-220,     y:= y1 + 50, typ:=1, rw1:=1, rw2:=1, h:= 40, hTxt:= 28),
            txt:=[548]       	// RND
			);
      r1o2_10  	: ARRAY[2..10] OF NH_OBJ_DAT :=
			[	(wh:=0),	// 2
            (wh:=0), //3
            (wh:=13, x:=50    , y:= y1+ 150,w:= x2-110  ,FgC := 4, BgC := 3 , fn := 2 ), 	//1 Interval generovnia
            (wh:=13, x:=50    , y:= y1+ 300,w:= x2-110  ,FgC := 4, BgC := 5 , fn := 3 ), 	//2 Min ON
            (wh:=13, x:=50    , y:= y1+ 400,w:= x2-110  ,FgC := 4, BgC := 6 , fn := 4 ), 	//3 Max ON
            (wh:=13, x:=50    , y:= y1+ 500,w:= x2-110  ,FgC := 4, BgC := 5 , fn := 5 ), 	//4 Min OFF
            (wh:=13, x:=50    , y:= y1+ 600,w:= x2-110  ,FgC := 4, BgC := 6 , fn := 6 ), 	//5 Max OFF
			 	(wh:=20, x:=70   , y:= y1+ 890,FgC :=13, w:=74, h := 72, cf :=(c:=3)), 			//9 Lock/Dark
			  	(wh:=20, x:=369  , y:= y1+ 730,FgC :=12, w:=48, h := 49, cf :=(c:=3))	];			//10 Daymode

		r2		: NH_DAYS_OF_WEEK;

      s  : ARRAY[0..6] OF NH_SLD_DAT :=
         [  (t:=1,v1:=1, v2:=31, fmt := '%3.0f', txt:= 116, zom:=0,tun:=0),        	// slider k start
				(t:=1,v1:=0, v2:=59, fmt := '%3.0f', txt:= 116, zom:=0,tun:=0),        	// nepouzije sa
            (t:=1, v2:=255,      fmt := 's%Tm:ss m'           , txt:= 538),
            (t:=3, v2:=600,      fmt := 'm%Th:mm h'           , txt:= 534),
            (t:=3, v2:=600,      fmt := 'm%Th:mm h'           , txt:= 535),
            (t:=3, v2:=600,      fmt := 'm%Th:mm h'           , txt:= 536),
            (t:=3, v2:=600,      fmt := 'm%Th:mm h'           , txt:= 537)
         ];
   END_STRUCT;

   NH_FRM_075 {HIDDEN}  :  STRUCT
      hed      : NH_FRM_HED := (Name:='_075',wht:=3);
      mnu      : NH_MNU := ( n:=3,                                  			// MNU-typovy den HOME
                        o := [
                              (fn :=   6,wh:=  6,cm :=  31),
                              (fn := 22),
										(fn := 273,wh:=274,cm := 205,x:=xc-45, frm:=76),		// typovy den
										(fn :=  20,wh:= 22,cm :=  22,x:=xc+45, frm:=0)			// zony
                           ]);
   END_STRUCT;

   NH_FRM_076   {HIDDEN}  :  STRUCT 	// HOME - centralne nastavenie typ.dnea
      hed      : NH_FRM_HED := (Name:='_076',desc:='FRM-HOME-typovy den',wht:=2,row:=3,sld:=2);
		r1  	: ARRAY[0..4] OF NH_OBJ_DAT :=
			[	(),
				(wh:=6, x:=xc, y:=y1+ 50,w:=500, h:=33,cf:=(n:=51), fgC:=4, fn:=2 ),	// 1; typovy den
				(wh:=6, x:=xc, y:=y1+330,w:=500,h:=28,cf:=(n:=553), fgC:=4, fn:=2 )	// 2; riadit sa kalendarom
			];
      r1_5_6_Type : NH_OBJ_123 :=                     			// rolovacii vyber - kedy prepnut na kalendar
      	(	wh:=123,cf:=(x:= 50,     y:= y1 + 390, typ:=1, rw1:=1, rw2:=10, h:= 41, hTxt:= 28),
            txt:=[206,207,208,209,210,211,212,213,214,215]
			);
		r1_7_9 	: ARRAY[7..9] OF NH_OBJ_DAT;             			// len volne riadky
		r1_10 	: ARRAY[10..10] OF NH_OBJ_DAT :=             			// len info parameter
      	      [(wh:= 6, x:=xc      , y:= 1015,       w:= 400, h:=20, Fgc:=2, fn:=2, nTch:=1, cf:=(c:=254))];  // 10 info dali nbr {len admin}

		r2_On	: NH_DAT_TIM2  := (txt:=                        	// zadanie datumu/casu
         [ (),(),(),(),(),(),(),(),
				(wh:=0),             										// ziadny text v urovni title
				(wh:=0)                         							// ziadny text pred datumom
			]);

		r3		: NH_DAYS_OF_WEEK  := (txt:=[( y:=y1+250, cf:=(c:=1), set6:=1 )]);

      s  	: ARRAY[0..1] OF NH_SLD_DAT :=
         [  (t:=1,v1:=1, v2:=31, fmt := '%3.0f', txt:= 116, zom:=0,tun:=0),        	// 0 slider k start
				(t := 5,v1:=1,       v2 := 1439.0  , fmt := ''          , txt :=   0, xv := x2-53, tun := 1  )                 // slider LUPY bodu, nevypisuje sa ani text, ani hodnota
         ];
   END_STRUCT;

   NH_FRM_077   {HIDDEN}  :  STRUCT 	// ROM - fazy dna rano-vecer
      hed      : NH_FRM_HED := (Name:='_077',wht:=2,row:=2,sld:=1);
		r1  	: ARRAY[0..10] OF NH_OBJ_DAT :=
			[	(wh:=0, w:=82, fn:=44, cm:=130), 																							// 0 obrazok kopirovania
				(wh:=6, x:=xc, y:=y1+ 60,w:=500, h:=33,cf:=(n:=555), fgC:=4, fn:=2 ),											// 1; text - faza dna
            (wh:=0, x:= x2- 70 , y:= y1 + 60,  w:= 62, Fn := 555,  FgC := 6, BgC := 50, h := 0, cf :=(c:=3)),  	// 2 prepinac obrazkov DayMode/On - vsetky obrazky na sebe (h:=0, cf.c>0)
				(),																																	// 3
            (wh:=14, x:= 50 ,    y:= y1 + 600, 	w:= x2-110, h := 200,  FgC := 4,  Fn := 315,prs:=0),     			// 4 OBJEKT slider day/evening/nighy/morning
            (wh:=0 , x:= 50,      					w:= x2-110 , FgC := 4,BgC := 5,  fn := 0, cm := 251)    				// 5 slider LUPY konkretneho bodu
			];

		r2	: NH_DAYS_OF_WEEK  := (txt:=[( y:=y1+300, cf:=(c:=1), set6:=1 )]);

      s  : ARRAY[0..0] OF NH_SLD_DAT :=
         [  (t := 5,v1:=1,       v2 := 1439.0  , fmt := ''          , txt :=   0, xv := x2-53, tun := 1  )                 // slider LUPY bodu, nevypisuje sa ani text, ani hodnota
         ];

   END_STRUCT;

   NH_FRM_078 {HIDDEN}  :  STRUCT
      hed      : NH_FRM_HED := (Name:='_078',wht:=3);
      mnu      : NH_MNU := ( n:=0,
	  							     o := [(
                                        fn :=  1, wh :=  1, cm := 25  ), //       // logo
                                       (fn := 23, wh := 25, cm := 250  ),         // setup
                                       (fn :=  3, wh :=  0, cm := 20   ),         // home
                                       (fn := 41, wh := 42, cm := 21   ),         // FAV
                                       (fn := 16, wh := 17, cm := 22   ),         // rom
                                       (fn := 10, wh := 11, cm := 23   ),         // cat
                                       (fn := 27, wh := 28, cm := 24   ),         // act
                                       (fn := 49, wh :=  0, cm := 26   )]         // ON/OFF
                           );
   END_STRUCT;
   NH_FRM_079 {HIDDEN}  :  STRUCT
      hed      : NH_FRM_HED := (Name:='_079',wht:=3);
      mnu      : NH_MNU := ( n:=0,
	  							     o := [		(fn :=  6, wh := 44, cm := 130, w:=72  ),  // sive/zlte copy
												//	(fn :=   6,wh:=  6,cm :=  31),
                                       (fn := 38, wh := 38, cm := 133, w:=72  ),  // zeleny check
                                       (fn :=  3, wh :=  0, cm := 20   ),         // home
                                       (fn := 41, wh := 42, cm := 21   ),         // FAV
                                       (fn := 16, wh := 17, cm := 22   ),         // rom
                                       (fn := 10, wh := 11, cm := 23   ),         // cat
                                       (fn := 27, wh := 28, cm := 24   ),         // act
                                       (fn := 49, wh :=  0, cm := 26   )]         // ON/OFF
                           );

   END_STRUCT;

   NH_FRM_080  {HIDDEN} :  STRUCT 	// Meteostanica - wind
      hed      : NH_FRM_HED := (Name:='_080',wht:=2,row:=1,sld:=11);
  		r0_10 : ARRAY[0..10] OF NH_OBJ_DAT :=
		  	[	(wh:=13, x:=50    , y:= y1+ 100,w:= x2-110  ,FgC := 4, BgC := 8 , fn := 0 ), 			//  0 slaby vietor
     			(wh:=13, x:=50    , y:= y1+ 180,w:= x2-110  ,FgC := 4, BgC :=18 , fn := 1 ), 			//  1 silny vietor
				(wh:=13, x:=50    , y:= y1+ 260,w:= x2-110  ,FgC := 4, BgC := 7 , fn := 2 ), 			//  2 kriticka rychlost

			  	(wh:=20, x:= x2-60, y:= y1+ 360,w:= 48     , FgC := 0, BgC :=50, fn := 567 ), 		//  3 manual
     			(wh:=13, x:=50    , y:= y1+ 460,w:= x2-110  ,FgC := 4, BgC := 3 , fn := 4 ), 			//  4 man-windspeed
            (wh:=13, x:=50    , y:= y1+ 540,w:= x2-110  ,FgC := 4, BgC := 3 , fn := 5 ), 			//  5 man-winddir
            (wh:=13, x:=50    , y:= y1+ 620,w:= x2-110  ,FgC := 4, BgC := 5 , fn := 6 ), 			//  6 man-spower

			  	(wh:=20, x:= x2-60, y:= y1+ 700,w:= 48   , FgC := 0, BgC :=50, fn := 578 ), 			//  7 posielat pre rolety
     			(wh:=13, x:=50    , y:= y1+ 800,w:= x2-110  ,FgC := 4, BgC := 3 , fn := 3 ), 			//  8 filt1r
     			(wh:=13, x:=50    , y:= y1+ 880,w:= x2-110  ,FgC := 4, BgC := 3 , fn := 7 ) 			//  9 WindSpeedRol

         ];
      s  : ARRAY[0..10] OF NH_SLD_DAT := [
				(		v2 := 50.0  , fmt := '%4.0f m/s', 	txt := 575, xv := x2-53 ),      			// 0 slaby vietor
				(		v2 := 50.0  , fmt := '%4.0f m/s', 	txt := 579, xv := x2-53 ),      			// 1 silny vietor
				(		v2 := 50.0  , fmt := '%4.0f m/s', 	txt := 576, xv := x2-53 ),     			// 2 kriticka rychost vetra
				(t:=3,v2 := 2000.0, fmt := '%4.0f', 		txt := 577, xv := x2-53 ), 				// 3 filter 1.r pre wietor
           	(		v2 := 50.0  , fmt := '%4.1f m/s', 	txt := 569, xv := x2-53,ink:=0.1 ),    // 4 man-rychlost vetra
				(t:=3,v2 := 360.0 , fmt := '%3.0f °', 		txt := 570, xv := x2-53 ), 				// 5 man-orientacia 360
				(		v2 := 1000.0, fmt := '%3.1f', 		txt := 571, xv := x2-53,ink:=0.1),      			// 6 man-spower
			 	(t:=1,v2 := 50.0  , fmt := '%4.0f m/s', 	txt := 606, xv := x2-53	)      			// 7 WindSpeedRol

         ];

   END_STRUCT;

   NH_FRM_081 {HIDDEN}  :  STRUCT
      hed      : NH_FRM_HED := (Name:='_081',wht:=3);
      mnu      : NH_MNU := ( n:=3,                                  				// MNU-ROL - submenu SETUP
                        o := [
                              (fn :=   6,wh:=  6,cm := 31),	// vrati sa na povodne menu
                              (fn := 114,wh:=114,cm :=31 ),
                              (fn := 119,wh:=115,cm := 205, frm:=65),   // parametre Up/Dn
                              (fn := 345,wh:=345,cm := 205, frm:=64),   // predvolby
                              (),
                              (),
                              (),
	                           (fn := 348,wh:=348,cm :=  82)        		// 7 Rom, ktore vstupuu do ZON

                           ]);
   END_STRUCT;

   NH_FRM_082 {HIDDEN}:  STRUCT 	// FRM-ROL - nastavit na poziciu
      hed      : NH_FRM_HED := (Name:='_082',wht:=2,row:=1,sld:=1,Desc:='FRM-ROL:Grafika');
		  	r1_0_4 	: ARRAY[0..4] OF NH_OBJ_DAT;
	   	r1_5_6 	: NH_OBJ_ROL;			// 2 riadky
		  	r1_7_10 	: ARRAY[7..10] OF NH_OBJ_DAT :=
		  	[	(wh:= 0, x:= 110, y:= y1 +826, 	w:= 150, h:=24, Fgc:=4, fn:=0, nTch:=1, cf:=(c:=254)),  				// 7 vypis realnej polohy yRol
				(wh:= 0, x:= 350, y:= y1 +826, 	w:= 150, h:=24, Fgc:=4, fn:=0, nTch:=1, cf:=(c:=254)),  				// 8 vypis realnej polohy yLam
            (wh:=13, x:= 50,  y:= y1 +900,  	w:= x2-110  ,FgC := 4, BgC := 5          , fn := 0             ),  // 9 s opozdenim
	         (wh:= 0, x:=xc  , y:= 1018, 		w:= 400, h:=20, Fgc:=2, fn:=2, nTch:=1, cf:=(c:=254)           )  // 10 info dali nbr {len admin}
    		];
      s  : ARRAY[0..0] OF NH_SLD_DAT :=
           [
            (t := 3, v2:=1800,      fmt := 's%Tm:ss m'           , txt:= 115)        // 6 opozdenie
              ];
   END_STRUCT;

   NH_FRM_083  {HIDDEN}  :  STRUCT 	// FRM - predolby teploty
      hed      : NH_FRM_HED := (Name:='_083',wht:=2,row:=1,sld:=3);
      r_0_3  : ARRAY[0..3] OF NH_OBJ_DAT :=
			[	(wh:=6, x:=xc, y:=y1+ 60,w:=500, h:=33,cf:=(n:=48), fgC:=4, fn:=2 ),							// 0; text nastavit predvolbu
				(wh:=0),
	         (wh:=22,x:=145,		y:=y1+150,fn:=1,cf:=(c:=4),h:=68,w:=48, cm:=251)                 // 3  auto/MAN, 0.1...3
			];
		WHT : NH_OBJ_123 :=            // r3
	 			(wh:=123,cf:=(x:= 160,    y:=y1+250, typ:=1, rw2:=3, h:= 50, hTxt:= 28),                     // 4+5 ON/OFF
    					txt:=[599,600]);
      r_6_10  : ARRAY[6..10] OF NH_OBJ_DAT :=
        [   (wh:=13, x:= 50     , y:= y1 + 500,   w:= x2-110 , FgC := 4, BgC := 3, fn := 0),       // 6 delay
            (wh:=13, x:= 50     , y:= y1 + 600,   w:= x2-110 , FgC := 4, BgC := 3, fn := 1),       // 7 wait
				(wh:=0),
				(wh:=0),
     	      (wh:= 6, x:=xc      , y:= 1020,       w:= 400, h:=20, Fgc:=2, fn:=2, nTch:=1, cf:=(c:=254))  // 10 info par {len admin}
        ];
      s  : ARRAY[0..2] OF NH_SLD_DAT := [
            ( t:=3, xv := x2-53, v2 := 3599.0 , fmt := 's%Tm:ss m',   txt:= 602),      // 0 s opozdenim
            ( t:=3, xv := x2-53, v2 := 3599.0 , fmt := 's%Tm:ss m',   txt:= 601)      // 1 ak bude trvat pohyb
         ];
   END_STRUCT;

   NH_FRM_084  {HIDDEN} :  STRUCT 	// Meteostanica - wind
      hed      : NH_FRM_HED := (Name:='_084',wht:=2,row:=1,sld:=11);
   	r1_0_1_Type : NH_OBJ_123 :=                     			// rolovacii vyber - kedy prepnut na kalendar
      	(	wh:=123,cf:=(x:= 50,     y:= y1 +  50, typ:=1, rw1:=1, rw2:=2, h:= 41, hTxt:= 28),
            txt:=[572,573,574]
			);
  		r1_2_10 : ARRAY[2..10] OF NH_OBJ_DAT :=
		  	[	(wh:=13, x:=50    , y:= y1+ 300,w:= x2-110  ,FgC := 4, BgC := 8 , fn := 0 ), 			//  2 nizka teplota
				(wh:=13, x:=50    , y:= y1+ 380,w:= x2-110  ,FgC := 4, BgC := 7 , fn := 1 ), 			//  3 vysoka teplota
     			(wh:=13, x:=50    , y:= y1+ 500,w:= x2-110  ,FgC := 4, BgC := 3 , fn := 2 ),			//  4 koef.ziarenia na osvetlenie
     			(wh:=13, x:=50    , y:= y1+ 580,w:= x2-110  ,FgC := 4, BgC := 3 , fn := 3 ), 			//  5 100% osvetlenie
     			(wh:=13, x:=50    , y:= y1+ 680,w:= x2-110  ,FgC := 4, BgC := 3 , fn := 4 ) 			//  6 FilsPower
         ];
      s  : ARRAY[0..10] OF NH_SLD_DAT := [
				(v1:=-10,v2 := 50.0  	,fmt := '%4.0f °', 		txt := 603, xv := x2-53  ),      		// 0 nizka teplota
				(			v2 := 50.0  	,fmt := '%4.0f °', 		txt := 295, xv := x2-53  ),      		// 1 vysoka teplota
				(v1:=1.0,v2 := 100.0  	,fmt := '%4.1f', 			txt := 605, xv := x2-53,ink:=0.1  ), 	// 2 koefTo100
				(t:=3,	v2 := 1000.0	,fmt := '%4.0f', 			txt := 604, xv := x2-53  ),     			// 3 100%  osvetlenia
				(t:=3,v2 := 2000.0, fmt := '%4.0f', 				txt := 577, xv := x2-53 ) 					// 4 FilsPower
         ];
   END_STRUCT;

   NH_FRM_085  {HIDDEN} :  STRUCT 	// Setup HET/VEN
      hed      : NH_FRM_HED := (Name:='_085',wht:=2,row:=1,sld:=11,desc:='Archivovat HET');
  		r0_10 : ARRAY[0..10] OF NH_OBJ_DAT :=
		  	[  (wh:=20, x:=x2-60 ,y:= y1 + 50, w:= 48     , 				FgC := 4, BgC :=50, 	fn := 100), //0 zablokovat
				(),
				(),
				(),
				(wh:=20, x:=x2-60 ,y:= y1 + 430, w:= 48     , 				FgC := 0, BgC :=50, 	fn := 615),	//  4 logovat
			   (wh:=20, x:=x2-60 ,y:= y1 + 480, w:= 48     , 				FgC := 0, BgC :=50, 	fn := 614),	//  5 kazda zmena Out
			  	(wh:=13, x:=50    , y:= y1+ 580,w:= x2-110  ,FgC := 4, BgC := 8 , fn := 0 ), 					//  6 sample
			  	(wh:=13, x:=50    , y:= y1+ 660,w:= x2-110  ,FgC := 4, BgC := 3 , fn := 1 ), 					//  7 ReQ
			  	(wh:=13, x:=50    , y:= y1+ 740,w:= x2-110  ,FgC := 4, BgC := 3 , fn := 2 ), 					//  8 Rom
			  	(wh:=13, x:=50    , y:= y1+ 820,w:= x2-110  ,FgC := 4, BgC := 3 , fn := 3 ), 					//  9 Het
			  	(wh:=13, x:=50    , y:= y1+ 900,w:= x2-110  ,FgC := 4, BgC := 3 , fn := 4 ) 					// 10 Kot
         ];
      s  : ARRAY[0..10] OF NH_SLD_DAT := [
				(t:=3, v1:=1.0,	v2 := 3599.0, fmt := 's%Tm:ss m', 			txt := 609, xv := x2-53 ), 				// 0 vzorka
				(t:=1, v1:=1.0,	v2 := 255.0,  fmt := '.%4.1f°', 			txt := 610, xv := x2-53 ), 					// 1 Zmena ReQ
				(t:=1, v1:=1.0,	v2 := 255.0,  fmt := '.%4.1f°', 			txt := 611, xv := x2-53 ), 					// 2 Zmena Rom
				(t:=1, v1:=1.0,	v2 := 255.0,  fmt := '.%4.1f°', 			txt := 612, xv := x2-53 ), 					// 3 Zmena Het
				(t:=2, v1:=1.0,	v2 := 255.0,  fmt := '.%4.1f°', 			txt := 613, xv := x2-53 ) 						// 4 ZmenaKot
         ];
   END_STRUCT;

   NH_FRM_086 {HIDDEN}:  STRUCT 	// HET-rozdiely teplot
      hed      : NH_FRM_HED := (Name:='_086',wht:=2,row:=1,sld:=2);
		r1_0_1 : ARRAY[0..1] OF NH_OBJ_DAT :=
         [	(wh:=6,  x:= x2/2  , y:= y1 + 60,   w:= 400    , FgC := 3, BgC := 0, fn := 2, h:=30,cf:=(n:=476)),  // 0
				(wh:=6,  x:= x2/2  , y:= y1 + 160,  w:= 400    , FgC := 4, BgC := 0, fn := 2, h:=30,cf:=(n:=477))  // 1
	   	]; 	// 0
      r1_2_3_Type : NH_OBJ_123 :=    			// rolovacii vyber - kedy prepnut na kalendar							// 2
      	(	wh:=123,cf:=(x:= 140,     y:= y1 + 220, typ:=1, rw1:=1, rw2:=2, h:= 41, hTxt:= 28),                       // 3
            txt:=[478,479] );
		r1_4_10 : ARRAY[4..10] OF NH_OBJ_DAT :=
      	[
            (wh:=14, x:= 50 ,    y:= y1 + 600, 	w:= x2-110, h := 200,  FgC := 4,  Fn := 315,prs:=0),     		// 4 OBJEKT slider day/evening/nighy/morning
            (wh:=0 , x:= 50,      					w:= x2-110 , FgC := 4,BgC := 5,  fn := 0, cm := 251),   			// 5 slider LUPY konkretneho bodu
			  	(wh:=13, x:=50    , y:= y1+ 850,w:= x2-110  ,FgC := 4, BgC := 3 , fn := 1 ), 								// 6 slider
				(wh:=0, x:= 50    , y:= y1 + 480,   w:= x2-110  ,FgC := 4, BgC := 2          , fn := 5             ), // 7 pv4
            (wh:=0, x:= 50    , y:= y1 + 830,   w:= x2-110  ,FgC := 4, BgC := 3          , fn := 7             ), // 8 pauza medzi predvolbami
            (wh:=0, x:= 50    , y:= y1 + 700,   w:= x2-110  ,FgC := 4, BgC := 3          , fn := 8             ), // 9 typ
            (wh:=0, x:= x2-60  , y:= y1 +  50,   w:= 48     , FgC := 0, BgC :=50          , fn := 246           ) //10 nastavit predvolenu poziciu
         ];

      s  : ARRAY[0..1] OF NH_SLD_DAT :=
         [  (t := 5, v1:=1.0,    v2 := 400.0  , fmt := ''          , txt :=   0, xv := x2-53, tun := 1  ),    // 0 slider LUPY bodu, nevypisuje sa ani text, ani hodnota
           (t := 3, v1:=1.0,    v2 := 1800.0  , fmt := 's%Tm:ss m' , txt := 609, xv := x2-53, tun := 1  )     // 1 odoberat vzorky
         ];

   END_STRUCT;

   NH_FRM_087 {HIDDEN}  :  STRUCT 	// MNU-VVO
      hed      : NH_FRM_HED := (Name:='_087',wht:=3,desc:='MNU: VVO');
      mnu      : NH_MNU := ( n:=5,
                        o := [
                              (fn :=   6,wh:=  6,cm :=  31),
                              (),
										(),
										(),
                              (fn := 23,wh:=25,cm := 205, frm:=70),      	// setup
										(fn:=348,wh:=348,cm :=  82   			)		  	// ROM->DEV
                           ]);
   END_STRUCT;

  	NH_FRM_088 {HIDDEN}:  STRUCT
      hed : NH_FRM_HED := (Name:='_088',wht:=2,row:=1,sld:=4,desc:='Par WSB/TLA/TGL');
  		r0_10 : ARRAY[0..10] OF NH_OBJ_DAT :=
			[	(wh:=6, x:=xc, y:=y1+ 50,w:=500, h:=30,cf:=(n:=123), fgC:=4, fn:=2 ),													// 0 text-nastavenie
            (wh:=13, x:= 50     , y:= y1 + 200,   w:= x2-110  ,FgC := 4, BgC := 3,  fn := 1            ), // 1 cakanie na dalsi click
            (wh:=13, x:= 50     , y:= y1 + 300,   w:= x2-110  ,FgC := 4, BgC := 3,  fn := 2            ), // 2 press
            (wh:=13, x:= 50     , y:= y1 + 400,   w:= x2-110  ,FgC := 4, BgC := 3,  fn := 3            ), // 3 hold
            (),
            (),
            (),
            (),
            (),
            (wh:=20,x:= x2-60  , y:= y1 + 800,   w:= 48     , FgC := 4, BgC :=50			  	, fn := 100	), 	// 9 zablokovat
            (wh:=0, x:= xc     , y:= y1 + 960,   w:=110,h:=20,FgC := 2, BgC := 0,  fn := 2, cf:=(c:=254))     // 10 cislo dsl/dlma
    		];
      s  : ARRAY[0..3] OF NH_SLD_DAT :=
           [
            (),                                                                    // 0
            (t := 1, v2 := 10.0    , fmt := '1%Ts.z s'           , txt:= 77),         // 1 cakanie na dalsi click
            (t := 1, v2 := 10.0    , fmt := '1%Ts.z s'           , txt:= 78),         // 2 press
            (t := 1, v2 := 20.0    , fmt := '1%Ts.z s'           , txt:= 79)          // 3 hold
           ];
   END_STRUCT;

  	NH_FRM_089 {HIDDEN}:  STRUCT
      hed : NH_FRM_HED := (Name:='_089',wht:=2,row:=1,sld:=0,desc:='TGL-Co zobrazit');
  		r0_0 : ARRAY[0..0] OF NH_OBJ_DAT :=
			[	(wh:=6, x:=xc, y:=y1+100,w:=500, h:=30,cf:=(n:=50), fgC:=4, fn:=2 ) ];													// 0 text-nastavenie
      r1_1_2_Type : NH_OBJ_123 :=    			// rolovacii vyber - kedy prepnut na kalendar							// 2
      	(	wh:=123,cf:=(x:= 100,  y:= y1 + 200, typ:=1, rw1:=1, rw2:=5, h:= 50, hTxt:= 28),                       // 3
			            txt:=[34,35,36,37,39] );
  		r0_3_10 : ARRAY[3..10] OF NH_OBJ_DAT;
   END_STRUCT;

  	NH_FRM_090 {HIDDEN}:  STRUCT
      hed : NH_FRM_HED := (Name:='_090',wht:=2,row:=1,sld:=0,desc:='Click/Akcia->WSB/TGL');
  		r0_7 : ARRAY[0..7] OF NH_OBJ_DAT :=
         [  (wh:= 10, x:= 110    , y:= y1 + 130,   w:= 190   , FgC := 1, BgC := 8, fn := 102, cm := 251),                       // 0 obrazok WSB
            (wh:=  8, x:= 260    , y:= y1 + 95,    w:= 70    , FgC := 1, BgC := 8, fn := 3, cf :=(c:=1,p:=35),fmt:='1' ),       // 1
            (wh:=  8, x:= 325    , y:= y1 + 95,    w:= 70    , FgC := 4, BgC := 0, fn := 3, cf :=(p:=35),fmt:='2' ),            // 2
            (wh:=  8, x:= 390    , y:= y1 + 95,    w:= 70    , FgC := 2, BgC := 0, fn := 3, cf :=(p:=35),fmt:='3' ),            // 3
            (wh:=  8, x:= 455    , y:= y1 + 95,    w:= 70    , FgC := 2, BgC := 0, fn := 3, cf :=(p:=35),fmt:='4' ),            // 4
            (wh:=  8, x:= 520    , y:= y1 + 95,    w:= 70    , FgC := 2, BgC := 0, fn := 3, cf :=(p:=35),fmt:='5' ),            // 5
            (wh:=  8, x:= 290    , y:= y1 +180,    w:= 90    , FgC := 8, BgC := 0, fn := 3, cf :=(p:=35),fmt:='Push' ),         // 6
            (wh:=  8, x:= 460    , y:= y1 +180,    w:= 90    , FgC := 2, BgC := 0, fn := 3, cf :=(p:=35),fmt:='Hold' )         // 7
			];
      r_8_9: NH_OBJ_123 :=    			// rolovacii vyber - kedy prepnut na kalendar							// 2
      	(	wh:=123,cf:=(x:= 100,  y:= y1 + 300, typ:=1, rw1:=1, rw2:=2, h:= 52, hTxt:= 28),                       // 3
//			            txt:=[80,181,180,179,182,188,189,178] );
			            txt:=[189,178] );
  		r_10 : ARRAY[10..10] OF NH_OBJ_DAT :=
            [(wh:=6,   x:=xc      , y:= 1015,       w:= 400, h:=20, Fgc:=2, fn:=2, nTch:=1, cf:=(c:=254) )];
   END_STRUCT;

   NH_FRM_091  {HIDDEN} :  STRUCT
      hed      : NH_FRM_HED := (Name:='_091',wht:=2,row:=1,sld:=0, desc:='Setup SCN');
  		r0_0 : ARRAY[0..0] OF NH_OBJ_DAT :=
			[	(wh:=6, x:=xc, y:=y1+80,w:=500, h:=30,cf:=(n:=621), fgC:=4, fn:=2 ) ];													// 0 text-nastavenie
      mnu   : NH_OBJ_123 := // R: 1..2
            (wh:=123,cf:=(x:= xc-200,     y:= y1 + 150, typ:=1, rw2:=3, h:= 50, hTxt:= 28),
                 txt:=[622,623,624]);                                                    // 1 rolovaci vyber textov
  		r3_3 : ARRAY[3..3] OF NH_OBJ_DAT :=
			[	(wh:=6, x:=xc, y:=y1+400,w:=500, h:=30,cf:=(n:=184), fgC:=4, fn:=2 ) ];													// 0 text-nastavenie
      r4_10   : ARRAY[4..10] OF NH_OBJ_DAT := [
				(),
				(),
            (),
            (),
            (wh:=20, x:= x2-140  , y:= y1 + 820,   w:= 48     , FgC := 0, BgC :=50          , fn := 228          ),  // 8 archivovat
            (wh:=20, x:= x2-140  , y:= y1 + 880,   w:= 48     , FgC := 4, BgC :=50          , fn := 100          ),  // 9 zablokovat
            (wh:= 6, x:=xc       , y:= 1015,       w:= 400, h:=20, Fgc:=2, fn:=2, nTch:=1, cf:=(c:=254)           )  // 10 info dali nbr {len admin}
             ];
   END_STRUCT;
   NH_FRM_092  {HIDDEN} :  STRUCT
      hed      : NH_FRM_HED := (Name:='_092',wht:=2,row:=1,sld:=0, desc:='Setup ACT');
  		r0_0 : ARRAY[0..0] OF NH_OBJ_DAT :=
			[	(wh:=6, x:=xc, y:=y1+80,w:=500, h:=30,cf:=(n:=620), fgC:=4, fn:=2 ) ];													// 0 text-nastavenie
      mnu   : NH_OBJ_123 := // R: 1..2
            (wh:=123,cf:=(x:= xc-200,     y:= y1 + 150, typ:=1, rw2:=3, h:= 50, hTxt:= 28),
                 txt:=[622,623,624]);                                                    // 1 rolovaci vyber textov
      r3_10   : ARRAY[3..10] OF NH_OBJ_DAT := [
				(wh:=0, x:=xc, y:=y1+100,w:=500, h:=30,cf:=(n:=50), fgC:=4, fn:=2 ),
				(),
				(),
            (),
            (),
            (wh:=20, x:= x2-140  , y:= y1 + 820,   w:= 48     , FgC := 0, BgC :=50          , fn := 228          ),  // 8 archivovat
            (wh:=20, x:= x2-140  , y:= y1 + 880,   w:= 48     , FgC := 4, BgC :=50          , fn := 100          ),  // 9 zablokovat
            (wh:= 6, x:=xc       , y:= 1015,       w:= 400, h:=20, Fgc:=2, fn:=2, nTch:=1, cf:=(c:=254)           )  // 10 info dali nbr {len admin}
             ];
   END_STRUCT;

   NH_FRM_093 {HIDDEN}  :  STRUCT
      hed      : NH_FRM_HED := (Name:='_093',wht:=3,desc:='Menu SCN');
      mnu      : NH_MNU := ( n:=3,
                        o := [
                              (fn :=   6,wh:=  6,cm :=  31),
                              (),
                              (fn :=  83,wh:= 84,cm := 205,x:=xc-90 	,frm:=9	),        // parametre
                              (fn :=  23,wh:= 24,cm := 205,x:=xc		,frm:=91	),        // setup
										(fn := 348,wh:=348,cm :=  82,x:=xc+90				)        // ROM ->
                           ]);
   END_STRUCT;

   NH_FRM_094 {HIDDEN}  :  STRUCT
      hed      : NH_FRM_HED := (Name:='_094',wht:=3,desc:='Menu ACT');
      mnu      : NH_MNU := ( n:=3,
                        o := [
                              (fn :=   6,wh:=  6,cm :=  31),
                              (),
                              (fn :=  23,wh:= 24,cm := 205,x:=xc-45	,frm:=92	),        // setup
										(fn := 348,wh:=348,cm :=  82,x:=xc+45				)        // ROM ->
                           ]);
   END_STRUCT;

END_TYPE

VAR_GLOBAL
//	yFrm_500	AT mObr			{HIDDEN} : NH_FRM_500;					// import from NH2.exp
//	yFrm_250	AT mObr			{HIDDEN} : NH_FRM_250;					// import from NH2.exp
//	yImp		AT yFrmData		{HIDDEN} : NH_LOG_IMP;					// only struct import
//   xFrmHed           		{HIDDEN} : PTR_TO NH_FRM_SAVE_MAP;  // head for saving

	// ladenie

END_VAR

	VAR_GLOBAL
   	xFrmHed           		{HIDDEN} : PTR_TO NH_FRM_SAVE_MAP;  // head for saving

	   _START_FRM_SYS : USINT := 0;

		_247_S : UDINT := SIZEOF(NH_FRM_247); _247 {PUBLIC} : NH_FRM_247 ;
   	_249_S : UDINT := SIZEOF(NH_FRM_249); _249 : NH_FRM_249 ;
   	_250_S : UDINT := SIZEOF(NH_FRM_250); _250 : NH_FRM_250 ;
   	_251_S : UDINT := SIZEOF(NH_FRM_251); _251 : NH_FRM_251 ;
   	_252_S : UDINT := SIZEOF(NH_FRM_252); _252 : NH_FRM_252 ;
   	_253_S : UDINT := SIZEOF(NH_FRM_253); _253 : NH_FRM_253 ;
   	_254_S : UDINT := SIZEOF(NH_FRM_254); _254 : NH_FRM_254 ;
   	_255_S : UDINT := SIZEOF(NH_FRM_255); _255 : NH_FRM_255 ;

		_500_S : UDINT := SIZEOF(NH_FRM_500); _500 : NH_FRM_500 ;
//   	_501_S : UDINT := SIZEOF(NH_LOG_HEAD); _501 : NH_LOG_HEAD := (hed:=(Name:='_501'));

	   _END_FRM_SYS    : UDINT := 0;

	   _START_FRM_WEB : USINT := 0;

		_000_S : UDINT := SIZEOF(NH_FRM_000); _000 : NH_FRM_000 ;   // 0 defult browser
	   _001_S : UDINT := SIZEOF(NH_FRM_001); _001 : NH_FRM_001 ;   // 1 FRM-1 DALI-M/S/ :   slidre HW-nastavenia
	   _002_S : UDINT := SIZEOF(NH_FRM_002); _002 : NH_FRM_002 ;   // 2 FRM-2 DALI-M :      TOOLS vymazat SHA, pridat NOVE SHA
	   _003_S : UDINT := SIZEOF(NH_FRM_003); _003 : NH_FRM_003 ;   // 3 BRW-dali-MASTERr
	   _004_S : UDINT := SIZEOF(NH_FRM_004); _004 : NH_FRM_004 ;
	   _005_S : UDINT := SIZEOF(NH_FRM_005); _005 : NH_FRM_005 ;
	   _006_S : UDINT := SIZEOF(NH_FRM_006); _006 : NH_FRM_006 ;
	   _007_S : UDINT := SIZEOF(NH_FRM_007); _007 : NH_FRM_007 ;
	   _008_S : UDINT := SIZEOF(NH_FRM_008); _008 : NH_FRM_008 ;
	   _009_S : UDINT := SIZEOF(NH_FRM_009); _009 : NH_FRM_009 ;
	   _010_S : UDINT := SIZEOF(NH_FRM_010); _010 : NH_FRM_010 ;
	   _011_S : UDINT := SIZEOF(NH_HOM_011); _011 : NH_HOM_011 ;
	   _012_S : UDINT := SIZEOF(NH_FRM_012); _012 : NH_FRM_012 ;
	   _013_S : UDINT := SIZEOF(NH_FRM_013); _013 : NH_FRM_013 ;
	   _014_S : UDINT := SIZEOF(NH_FRM_014); _014 : NH_FRM_014 ;
	   _015_S : UDINT := SIZEOF(NH_FRM_015); _015 : NH_FRM_015 ;
	   _016_S : UDINT := SIZEOF(NH_FRM_016); _016 : NH_FRM_016 ;
   	_017_S : UDINT := SIZEOF(NH_FRM_017); _017 : NH_FRM_017 ;
	   _018_S : UDINT := SIZEOF(NH_FRM_018); _018 : NH_FRM_018 ;
   	_019_S : UDINT := SIZEOF(NH_FRM_019); _019 : NH_FRM_019 ;
	   _020_S : UDINT := SIZEOF(NH_FRM_020); _020 : NH_FRM_020 ;
   	_021_S : UDINT := SIZEOF(NH_FRM_021); _021 : NH_FRM_021 ;
	   _022_S : UDINT := SIZEOF(NH_FRM_022); _022 : NH_FRM_022 ;
   	_023_S : UDINT := SIZEOF(NH_FRM_023); _023 : NH_FRM_023 ;
   	_024_S : UDINT := SIZEOF(NH_FRM_024); _024 : NH_FRM_024 ;
	   _025_S : UDINT := SIZEOF(NH_FRM_025); _025 : NH_FRM_025 ;
	   _026_S : UDINT := SIZEOF(NH_FRM_026); _026 : NH_FRM_026 ;
 	  	_027_S : UDINT := SIZEOF(NH_FRM_027); _027 : NH_FRM_027 ;
	   _028_S : UDINT := SIZEOF(NH_FRM_028); _028 : NH_FRM_028 ;
   	_029_S : UDINT := SIZEOF(NH_FRM_029); _029 : NH_FRM_029 ;
	   _030_S : UDINT := SIZEOF(NH_FRM_030); _030 : NH_FRM_030 ;
   	_031_S : UDINT := SIZEOF(NH_FRM_031); _031 : NH_FRM_031 ; 		//31 FRM - ROM*set typ miestnosti
	   _032_S : UDINT := SIZEOF(NH_FRM_032); _032 : NH_FRM_032 ;
   	_033_S : UDINT := SIZEOF(NH_FRM_033); _033 : NH_FRM_033 ;
	   _034_S : UDINT := SIZEOF(NH_FRM_034); _034 : NH_FRM_034 ;
   	_035_S : UDINT := SIZEOF(NH_FRM_035); _035 : NH_FRM_035 ;
	   _036_S : UDINT := SIZEOF(NH_FRM_036); _036 : NH_FRM_036 ;
   	_037_S : UDINT := SIZEOF(NH_FRM_037); _037 : NH_FRM_037 ;
	   _038_S : UDINT := SIZEOF(NH_FRM_038); _038 : NH_FRM_038 ;
   	_039_S : UDINT := SIZEOF(NH_FRM_039); _039 : NH_FRM_039 ;
	   _040_S : UDINT := SIZEOF(NH_FRM_040); _040 : NH_FRM_040 ;
   	_041_S : UDINT := SIZEOF(NH_FRM_041); _041 : NH_FRM_041 ;
	   _042_S : UDINT := SIZEOF(NH_FRM_042); _042 : NH_FRM_042 ;
   	_043_S : UDINT := SIZEOF(NH_FRM_043); _043 : NH_FRM_043 ;
	   _044_S : UDINT := SIZEOF(NH_FRM_044); _044 : NH_FRM_044 ;
   	_045_S : UDINT := SIZEOF(NH_FRM_045); _045 : NH_FRM_045 ;
	   _046_S : UDINT := SIZEOF(NH_FRM_046); _046 : NH_FRM_046 ;
   	_047_S : UDINT := SIZEOF(NH_FRM_047); _047 : NH_FRM_047 ;
	   _048_S : UDINT := SIZEOF(NH_FRM_048); _048 : NH_FRM_048 ;
   	_049_S : UDINT := SIZEOF(NH_FRM_049); _049 : NH_FRM_049 ;
	   _050_S : UDINT := SIZEOF(NH_FRM_050); _050 : NH_FRM_050 ;
   	_051_S : UDINT := SIZEOF(NH_FRM_051); _051 : NH_FRM_051 ;
	   _052_S : UDINT := SIZEOF(NH_FRM_052); _052 : NH_FRM_052 ;
   	_053_S : UDINT := SIZEOF(NH_FRM_053); _053 : NH_FRM_053 ;
	   _054_S : UDINT := SIZEOF(NH_FRM_054); _054 : NH_FRM_054 ;
   	_055_S : UDINT := SIZEOF(NH_FRM_055); _055 : NH_FRM_055 ;
	   _056_S : UDINT := SIZEOF(NH_FRM_056); _056 : NH_FRM_056 ;
  	   _057_S : UDINT := SIZEOF(NH_FRM_057); _057 : NH_FRM_057 ;      // TGL-display
	   _058_S : UDINT := SIZEOF(NH_FRM_058); _058 : NH_FRM_058 ;
   	_059_S : UDINT := SIZEOF(NH_FRM_059); _059 : NH_FRM_059 ;
	   _060_S : UDINT := SIZEOF(NH_FRM_060); _060 : NH_FRM_060 ;
   	_061_S : UDINT := SIZEOF(NH_FRM_061); _061 : NH_FRM_061 ;
	   _062_S : UDINT := SIZEOF(NH_FRM_062); _062 : NH_FRM_062 ;
   	_063_S : UDINT := SIZEOF(NH_FRM_063); _063 : NH_FRM_063 ;
	   _064_S : UDINT := SIZEOF(NH_FRM_064); _064 : NH_FRM_064 ;
   	_065_S : UDINT := SIZEOF(NH_FRM_065); _065 : NH_FRM_065 ;
	   _066_S : UDINT := SIZEOF(NH_FRM_066); _066 : NH_FRM_066 ;
   	_067_S : UDINT := SIZEOF(NH_FRM_067); _067 : NH_FRM_067 ;
	   _068_S : UDINT := SIZEOF(NH_FRM_068); _068 : NH_FRM_068 ;
	   _069_S : UDINT := SIZEOF(NH_FRM_069); _069 : NH_FRM_069 ;
   	_070_S : UDINT := SIZEOF(NH_FRM_070); _070 : NH_FRM_070 ;
	   _071_S : UDINT := SIZEOF(NH_FRM_071); _071 : NH_FRM_071 ;
   	_072_S : UDINT := SIZEOF(NH_FRM_072); _072 : NH_FRM_072 ;
	   _073_S : UDINT := SIZEOF(NH_FRM_073); _073 : NH_FRM_073 ;
   	_074_S : UDINT := SIZEOF(NH_FRM_074); _074 : NH_FRM_074 ;
	   _075_S : UDINT := SIZEOF(NH_FRM_075); _075 : NH_FRM_075 ;
   	_076_S : UDINT := SIZEOF(NH_FRM_076); _076 : NH_FRM_076 ;
	   _077_S : UDINT := SIZEOF(NH_FRM_077); _077 : NH_FRM_077 ;
   	_078_S : UDINT := SIZEOF(NH_FRM_078); _078 : NH_FRM_078 ;
	   _079_S : UDINT := SIZEOF(NH_FRM_079); _079 : NH_FRM_079 ;
   	_080_S : UDINT := SIZEOF(NH_FRM_080); _080 : NH_FRM_080 ;
	   _081_S : UDINT := SIZEOF(NH_FRM_081); _081 : NH_FRM_081 ;
   	_082_S : UDINT := SIZEOF(NH_FRM_082); _082 : NH_FRM_082 ;
		_083_S : UDINT := SIZEOF(NH_FRM_083); _083 : NH_FRM_083 ;
	   _084_S : UDINT := SIZEOF(NH_FRM_084); _084 : NH_FRM_084 ;
   	_085_S : UDINT := SIZEOF(NH_FRM_085); _085 : NH_FRM_085 ;
	   _086_S : UDINT := SIZEOF(NH_FRM_086); _086 : NH_FRM_086 ;
	   _087_S : UDINT := SIZEOF(NH_FRM_087); _087 : NH_FRM_087 ;
	   _088_S : UDINT := SIZEOF(NH_FRM_088); _088 : NH_FRM_088 ;
	   _089_S : UDINT := SIZEOF(NH_FRM_089); _089 : NH_FRM_089 ;
	   _090_S : UDINT := SIZEOF(NH_FRM_090); _090 : NH_FRM_090 ;
	   _091_S : UDINT := SIZEOF(NH_FRM_091); _091 : NH_FRM_091 ;
	   _092_S : UDINT := SIZEOF(NH_FRM_092); _092 : NH_FRM_092 ;
	   _093_S : UDINT := SIZEOF(NH_FRM_093); _093 : NH_FRM_093 ;
	   _094_S : UDINT := SIZEOF(NH_FRM_094); _094 : NH_FRM_094 ;
